(* CODESYS project sortingmachineOOP

Project tree, tasks and I/O mapping:
  Device : CODESYS Control Win V3 x64, 3S - Smart Software Solutions GmbH, version 3.5.16.40
    application Application
      libraries: Standard, * (System); Util, * (System); OMAC PackML State Machine, 1.0.0.4 (3S - Smart Software Solutions GmbH); Alarm Manager Interfaces, * (Intern); SysTypes Interfaces, 3.5.2.0 (System); VisuDialogs, * (System); XML parsing and composing library, * (Open Source); StringUtils, 3.5.17.0 (System); SysMem, 3.5.17.0 (System); CAA File, 3.5.17.0 (CAA Technical Workgroup); CAA Types Extern, 3.5.17.0 (CAA Technical Workgroup); CmpErrors Interfaces, * (System); SysDir, 3.5.17.0 (System); SysFile, 3.5.17.0 (System); SysTimeRtc, 3.5.17.0 (System)
      task AlarmManagerTask (cyclic, interval 50 ms, priority 31) calls AlarmManager.Alarm_Prg
      task MainTask (cyclic, interval t#20ms, priority 1) calls PLC_PRG, Sortery, LogowanieDanych
      task Task (cyclic, interval 5 ms, priority 1) calls POU_cyclic
      task VISU_TASK (cyclic, interval 100 ms, priority 31) calls VisuElems.Visu_Prg
      Alarm Configuration
        alarm group AlarmGroup1
            0 [Error]: Comparison Equal, ExpressionToCompare FALSE, Expression FIO.xEmergencyStop - "Przycisk bezpieczeństwa"
            2 [Warning]: Comparison Equal, ExpressionToCompare TRUE, Expression FIO.xSyrena - "Koniec przerwy"
            3 [Info]: Comparison Equal, ExpressionToCompare PACK_ML.State.Held, Expression PLC_PRG.unitModeManager.ActiveUnitMode.CurrentState - "Maszyna w stanie HELD"
            4 [Info]: Comparison Equal, ExpressionToCompare PACK_ML.State.Suspended, Expression PLC_PRG.unitModeManager.ActiveUnitMode.CurrentState - "Maszyna w stanie SUSPENDED"
            5 [Error]: Comparison Equal, ExpressionToCompare PACK_ML.State.Aborted, Expression PLC_PRG.unitModeManager.ActiveUnitMode.CurrentState - "Maszyna w stanie ABORTED"
        text list AlarmGroup1
        alarm group AlarmGroup2
        text list AlarmGroup2
        alarm group AlarmGroup3
        text list AlarmGroup3
        text list AlarmGroup
        AlarmStorage
        alarm class Error (priority 10, acknowledge ACK_REP_ACK)
        alarm class Info (priority 100, acknowledge REP)
        alarm class Warning (priority 30, acknowledge REP_ACK)
      Alarmy/
        function block AlarmFilterCriteria [ST]: AreAllAlarmClassesSelected, AreAllAlarmGroupsSelected, GetAlarmClasses, GetAlarmGroups, GetCountAlarmClasses, GetCountAlarmGroups, GetPriorityFrom, GetPriorityTo
        function block AlarmManagerClient [ST]: ActiveAlarmsChanged, AfterInit, AlarmStorageModified, GetFilterCriteria
        function ProcessAlarms [ST]
        data type StructureAlarmAsStrings
      Class Diagram
      Czas/
        function PobranieCzasu [ST]
        function UpdateEventTimestampWithSystemTime [ST]
      Data logger/
        data type E_EventSeverity
        data type E_EventType
        data type E_MaxString
        function block FB_CsvPersistentEventStorage [ST]: CreateCsvString, StoreEvent
        function block FB_EventLogger [ST]: AddEvent, FB_Init, IsEventBufferFull
        function block FB_XmlPac [ST]: ComposeXmlExample, FB_Init, OpenWriteClose, Parse, StoreEvent
        data type ST_Event
      data type eKolumnaKolor
      Interfejsy/
        interface I_Kolumna: M_BuzzerOnOff, M_UstawKolor
        interface I_PersistentEventStorage: StoreEvent
        interface I_Przenosnik: MaxPredkosc, MinPredkosc, PredkoscZadana, Start, Stop
      Obiekty/
        function block FB_Kolumna [ST]: M_BuzzerOnOff, M_UstawKolor
        function block FB_Przenosnik [ST]: MaxPredkosc, MinPredkosc, Predkosc, PredkoscZadana, Start, Stop
        function block FB_PrzenosnikNowy [ST]: AktualnaLiczbaZleconychProduktow, ZlecenieProdukty, ZliczajProdukty
        function block Sorter [ST]
        function block Sorter_1 [ST]: Bazowanie, Bazowanie_koniec, Czekaj, Error, FB_Init, Init, Sortowanie, SortowanieKoniec, TRANS_BAZOWANIE, TRANS_BAZOWANIE_KONIEC, TRANS_CZEKAJ, TRANS_ERROR, TRANS_INIT, TRANS_SORTOWANIE, TRANS_SORTOWANIE_KONIEC
      visualisation Panel
      Programy/
        program LogowanieDanych [ST]
        program PLC_PRG [ST]
        program POU_cyclic [ST]
        program Sortery [ST]
      Zmienne globalne/
        global variables FIO
        global variables GVL
    Ethernet : Ethernet, 3S - Smart Software Solutions GmbH, version 3.5.17.0
      Modbus_TCP_Master : Modbus TCP Master, 3S - Smart Software Solutions GmbH, version 3.5.16.0
          settings: AutoReconnect = TRUE
        Modbus_TCP_Slave : Modbus TCP Slave, 3S - Smart Software Solutions GmbH, version 3.5.16.0
            settings: Unit-ID = 1; IPAddress = [127, 0, 0, 1]; Salon_A_FC_02.Function Code = 2; Salon_A_FC_02.Read Offset = 16#0000; Salon_A_FC_02.Read Length = 16; Salon_A_FC_02.Write Offset = 0; Salon_A_FC_02.Write Length = 0; Salon_A_FC_02.Cycle Time = 100; Salon_A_FC_03.Function Code = 4; Salon_A_FC_03.Read Offset = 16#0000; Salon_A_FC_03.Read Length = 8; Salon_A_FC_03.Write Offset = 0; Salon_A_FC_03.Write Length = 0; Salon_A_FC_03.Cycle Time = 20; Salon_A_FC_15.Function Code = 15; Salon_A_FC_15.Read Offset = 0; Salon_A_FC_15.Read Length = 0; Salon_A_FC_15.Write Offset = 16#0000; Salon_A_FC_15.Write Length = 16; Salon_A_FC_15.Cycle Time = 100; Channel 3.Function Code = 16; Channel 3.Read Offset = 0; Channel 3.Read Length = 0; Channel 3.Write Offset = 16#0000; Channel 3.Write Length = 5; Channel 3.Cycle Time = 100
            input  Application.FIO.xPrzyciskStart : BOOL  // Salon_A_FC_02.Salon_A_FC_02.Bit0
            input  Application.FIO.xPrzyciskStop : BOOL  // Salon_A_FC_02.Salon_A_FC_02.Bit1
            input  Application.FIO.xPrzyciskReset : BOOL  // Salon_A_FC_02.Salon_A_FC_02.Bit2
            input  Application.FIO.xEmergencyStop : BOOL  // Salon_A_FC_02.Salon_A_FC_02.Bit3
            input  Application.FIO.xTrybAutoManual : BOOL  // Salon_A_FC_02.Salon_A_FC_02.Bit4
            input  Application.FIO.xCzujnikWejscie : BOOL  // Salon_A_FC_02.Salon_A_FC_02.Bit5
            input  Application.FIO.xCzujnikElementNOK_1 : BOOL  // Salon_A_FC_02.Salon_A_FC_02.Bit6
            input  Application.FIO.xCzujnikElementOK_2 : BOOL  // Salon_A_FC_02.Salon_A_FC_02.Bit7
            input  Application.FIO.xCzujnikElementOK_3 : BOOL  // Salon_A_FC_02.Salon_A_FC_02.Bit0
            input  Application.FIO.xFIOAktywny : BOOL  // Salon_A_FC_02.Salon_A_FC_02.Bit1
            input  Application.FIO.iCzujnikWizyjny : WORD  // Salon_A_FC_03.Salon_A_FC_03
            output Application.FIO.xLampkaStart : BOOL  // Salon_A_FC_15.Salon_A_FC_15.Bit0
            output Application.FIO.xLampkaStop : BOOL  // Salon_A_FC_15.Salon_A_FC_15.Bit1
            output Application.FIO.xLampkaReset : BOOL  // Salon_A_FC_15.Salon_A_FC_15.Bit2
            output Application.FIO.xSorterObroc_1 : BOOL  // Salon_A_FC_15.Salon_A_FC_15.Bit3
            output Application.FIO.xSorterPas_1 : BOOL  // Salon_A_FC_15.Salon_A_FC_15.Bit4
            output Application.FIO.xSorterObroc_2 : BOOL  // Salon_A_FC_15.Salon_A_FC_15.Bit5
            output Application.FIO.xSorterPas_2 : BOOL  // Salon_A_FC_15.Salon_A_FC_15.Bit6
            output Application.FIO.xSorterObroc_3 : BOOL  // Salon_A_FC_15.Salon_A_FC_15.Bit7
            output Application.FIO.xSorterPas_3 : BOOL  // Salon_A_FC_15.Salon_A_FC_15.Bit0
            output Application.FIO.xPrzeslona : BOOL  // Salon_A_FC_15.Salon_A_FC_15.Bit1
            output Application.FIO.xKolumnaLampaCzerwona : BOOL  // Salon_A_FC_15.Salon_A_FC_15.Bit2
            output Application.FIO.xKolumnaLampaZielona : BOOL  // Salon_A_FC_15.Salon_A_FC_15.Bit3
            output Application.FIO.xKolumnaLampaZolta : BOOL  // Salon_A_FC_15.Salon_A_FC_15.Bit4
            output Application.FIO.xKolumnaLampaNiebieski : BOOL  // Salon_A_FC_15.Salon_A_FC_15.Bit5
            output Application.FIO.xEmiter : BOOL  // Salon_A_FC_15.Salon_A_FC_15.Bit6
            output Application.FIO.xSyrena : BOOL  // Salon_A_FC_15.Salon_A_FC_15.Bit7
            output Application.FIO.iPodajnikWejsciowy : WORD  // Channel 3.Channel 3
            output Application.FIO.iPodajnikWyjsciowy : WORD  // Channel 3.Channel 3
            output Application.FIO.iLicznik_1 : WORD  // Channel 3.Channel 3
            output Application.FIO.iLicznik_2 : WORD  // Channel 3.Channel 3
            output Application.FIO.iLicznik_3 : WORD  // Channel 3.Channel 3
            unmapped channels: Salon_A_FC_02, Salon_A_FC_03, Salon_A_FC_15, Channel 3
  text list GlobalTextList
*)

// Device/Application/eKolumnaKolor
{attribute 'qualified_only'}
{attribute 'strict'}
TYPE eKolumnaKolor :
(
	zielony := 0,
	czerwony := 1,
	zolty := 2,
	niebieski := 3
);
END_TYPE

// Device/Application/Alarmy/StructureAlarmAsStrings
/// This structure contains the data the alarm table simulation displays in one row
TYPE StructureAlarmAsStrings :
STRUCT
	sState		: STRING;
	sID			: STRING;
	sInternalID	: STRING;
	sMessage	: STRING;
	sAlarmGroup	: STRING;
	sTSLast		: STRING;
	sAlarmClass	: STRING;
	sPriority	: STRING;
	sCurrValue	: STRING;
	sLatchVar1	: STRING;
	sLatchVar2	: STRING;
END_STRUCT
END_TYPE

// Device/Application/Data logger/E_EventSeverity
{attribute 'qualified_only'}
{attribute 'strict'}
TYPE E_EventSeverity :
(
    Verbose  := 0, // in progress
    Info     := 1, 
    Warning  := 2, 
    Error    := 3, 
    Critical := 4);
END_TYPE

// Device/Application/Data logger/E_EventType
{attribute 'qualified_only'}
{attribute 'strict'}
{attribute 'to_string'}
TYPE E_EventType :
(
	Alarm := 0,
	Message := 1
);
END_TYPE

// Device/Application/Data logger/E_MaxString
{attribute 'qualified_only'}
{attribute 'strict'}
TYPE E_MaxString :
(
	MaxString := 255
);
END_TYPE

// Device/Application/Data logger/ST_Event
TYPE ST_Event :
STRUCT
	eEventType : E_EventType;
	eEventSeverity: E_EventSeverity;
	nEventIdentity : UDINT;
	sEventText : STRING(255);
	dtTimeStamp: DATE_AND_TIME;
END_STRUCT

END_TYPE

// Device/Application/Zmienne globalne/FIO
{attribute 'qualified_only'}
VAR_GLOBAL
	(* zmienne wejściowe *)
	xPrzyciskStart:BOOL; // Start przenośnika - wejście PLC
	xPrzyciskStop:BOOL; // Stop przenośnika - wejście PLC
	xPrzyciskReset: BOOL; // Reset maszyny
	xEmergencyStop: BOOL; // Stop awaryjny
	xTrybAutoManual: BOOL; // Przełącznik piórkowy, mtryb auto/manual
	xCzujnikWejscie: BOOL; // czujnik na linii wejściowej
	xCzujnikElementNOK_1: BOOL; // wykrywa elementy wadliwe na linii, zsuwnia pierwsza
	xCzujnikElementOK_2: BOOL; // wykrywa elementy poprawne, zsuwnia druga
	xCzujnikElementOK_3: BOOL; //  wykrywa elementy poprawne, zsuwnia trzecia
	xFIOAktywny: BOOL;
	
	
	iCzujnikWizyjny: INT; // zwraca wartości ID poszczególnych elementów na linii
	
	(* zmienne wyjściowe *)
	xLampkaStart:BOOL; // podświetlenie przycisku start
	xLampkaStop:BOOL; // podśwoetlenie przycisku stop
	xLampkaReset: BOOL; // podśwoetlenie przycisku reet
	xSorterObroc_1: BOOL; // sorter spychający wadliwe elementy do zsuwni, sorter 1
	xSorterPas_1: BOOL; // pas sortera nr 1
	xSorterObroc_2: BOOL; // sorter spychający prawidłowe elementy do zsuwni, sorter 2
	xSorterPas_2: BOOL; // pas sortera nr 2
	xSorterObroc_3: BOOL; // sorter spychający prawidłowe elementy do zsuwni, sorter 3
	xSorterPas_3: BOOL; // pas sortera nr 3
	xPrzeslona: BOOL; // przesłona między podajnikami
	xSyrena:BOOL; // Syrena na przenośniku
	xKolumnaLampaCzerwona: BOOL; //  czerwona lampa kolumna świetlna
	xKolumnaLampaZielona: BOOL; //  zielona lampa kolumna świetlna
	xKolumnaLampaZolta: BOOL; //  zółta lampa kolumna świetlna
	xKolumnaLampaNiebieski : BOOL; //  niebeiska lampka kolumna świetlna
	xSorterLampa_1 :BOOL; // sygnalizacja świetlna sortera nr 1
	xSorterLampa_2 :BOOL; // sygnalizacja świetlna sortera nr 2
	xSorterLampa_3 :BOOL; // sygnalizacja świetlna sortera nr 3
	xEmiter: bool; // generator elementów na liniii
	
	iPodajnikWejsciowy: INT; // wpisujemy wartośc od 0-1000 w celu regulacji prędkości podajnika
	iPodajnikWyjsciowy: INT; // wpisujemy wartośc od 0-1000 w celu regulacji prędkości podajnika
	iLicznik_1: INT; 
	iLicznik_2: INT;
	iLicznik_3: INT;

END_VAR

// Device/Application/Zmienne globalne/GVL
{attribute 'qualified_only'}
VAR_GLOBAL
	xErrorActive:BOOL:=0;
	aAlarmy: ARRAY [0..19] OF BOOL; 	// tablica alarmów, klasa Error
	wAlarmy: WORD:=0;
	xResetAlarm: BOOL;
	g_sAlarmID:STRING;
    aRejestrProduktow : ARRAY[0..100] OF DINT;
    diSensorWizyjnyOstatniaWartosc : DINT;
    xLiniaStart : BOOL;
    xAlarmAktywny : BOOL;
	R_TRIG_Start:R_TRIG;
	R_TRIG_Reset:F_TRIG; 
	g_sMainDirectory : STRING := 'c:/'; // ścieżka głowna pliku CSV dla data logger
END_VAR
VAR_GLOBAL CONSTANT
	{attribute 'const_replaced'}
	gc_iNoOfCollumns:INT :=15;
	gc_iLengthOfDataArray:INT:=255;
	
	// PackML
	gc_sPRODUCTION : STRING := 'Production';
	gc_sSEMIAUTO : STRING := 'Semi Auto';
	gc_sSETUP : STRING := 'Setup';
END_VAR

// Device/Application/Programy/PLC_PRG
PROGRAM PLC_PRG
VAR
	productionUnitMode	: PACK_ML.UnitMode; // Example unit mode for prodction
	semiAutoUnitMode	: PACK_ML.UnitMode; // Example unit mode for semi auto production
	setupUnitMode		: PACK_ML.UnitMode; // Example unit mode for setup
	unitModeManager		: PACK_ML.UnitModeManager; // Unit mode manager to switch between unitmodes
	currentUnitMode		: PACK_ML.IUnitMode;
	xInit				: BOOL := FALSE; // Flag for initialization	
	
	// Visu Commands	
	xAbort				: BOOL;
	xActingStateComplete: BOOL;
	xClear				: BOOL;
	xHold				: BOOL;
	xReset				: BOOL;
	xStart				: BOOL;
	xStop				: BOOL;
	xSuspend			: BOOL;
	xUnHold				: BOOL;
	xUnSuspend			: BOOL;
	
	// Helper
	xSimulate			: BOOL;
	xChangeState		: BOOL := FALSE;	
	timer1				: TON;	
	iSelectedUnitMode	: INT := 0;
	iLastSelectedUnitMode: INT := 0;
	xUserModeChanged	: BOOL;
	xTest: BOOL;
	itest: INT;
	
	fbPrzenosnik: FB_PrzenosnikNowy;
	
	// alarm manager
	mAlarmManagerClient: AlarmManagerClient;
	
	StartStop: RS;
	xZlecenieWykonane: BOOL;
	LicznikElementyNaLinii: CTUD;
	iMaxPredkosc_visu: INT;
	iMinPredkosc_visu: INT;
	iPredkoscZadana_visu: INT;
	iZlecenie_visu: INT;
	xPotwierdzParametry_visu: BOOL;
	
	fbRtrigCzujnikSorter_1: r_trig;
	fbRtrigCzujnikSorter_2: r_trig;
	fbRtrigCzujnikSorter_3: r_trig;
	xResetZlecenie_visu: BOOL;
	iAktualnaLiczbaZleconychProduktow_visu: INT;
	fbKolumna: FB_Kolumna;
END_VAR

// inicjalizacja trybu pracy w standardzie Pack ML
IF NOT xInit THEN
	productionUnitMode(		sName := gvl.gc_sPRODUCTION, 
							dwSupportedStates := PACK_ML.State.All, 
							dwAllowsLeavingFromStates := PACK_ML.State.Stopped OR PACK_ML.State.Aborted OR PACK_ML.State.Idle, 
							dwAllowsEnteringIntoStates := PACK_ML.State.Stopped OR PACK_ML.State.Aborted OR PACK_ML.State.Idle, 
							eInitialState := PACK_ML.State.Resetting,
							xActive := TRUE);
	semiAutoUnitMode(		sName := gvl.gc_sSEMIAUTO, 
							dwSupportedStates := PACK_ML.State.All - PACK_ML.State.Completing - PACK_ML.State.Complete - PACK_ML.State.Holding - PACK_ML.State.Held - PACK_ML.State.UnHolding,
							dwAllowsLeavingFromStates := PACK_ML.State.Stopped OR PACK_ML.State.Aborted OR PACK_ML.State.Idle, 
							dwAllowsEnteringIntoStates := PACK_ML.State.Stopped OR PACK_ML.State.Aborted OR PACK_ML.State.Idle,   
							eInitialState := PACK_ML.State.Idle, 
							xActive := FALSE);
	setupUnitMode(			sName := gvl.gc_sSETUP, 
							dwSupportedStates := PACK_ML.State.All - PACK_ML.State.Completing - PACK_ML.State.Complete - PACK_ML.State.Holding - PACK_ML.State.Held - PACK_ML.State.UnHolding - PACK_ML.State.UnSuspending - PACK_ML.State.Suspended - PACK_ML.State.Suspending,
							dwAllowsLeavingFromStates := PACK_ML.State.Stopped OR PACK_ML.State.Aborted OR PACK_ML.State.Idle,   
							dwAllowsEnteringIntoStates := PACK_ML.State.Stopped OR PACK_ML.State.Aborted OR PACK_ML.State.Idle, 
							eInitialState := PACK_ML.State.Idle, 
							xActive := FALSE);
	
	// inicjalizacja wartości dla maszyny
	fbPrzenosnik.MaxPredkosc := 10;
	fbPrzenosnik.MinPredkosc := 2;
	fbPrzenosnik.PredkoscZadana := 4;
			

	// Register the unit modes 
	unitModeManager.Register(productionUnitMode);
	unitModeManager.Register(semiAutoUnitMode);
	unitModeManager.Register(setupUnitMode);
	xInit := TRUE;
END_IF

IF FIO.xFIOAktywny THEN
	
mAlarmManagerClient();

fbKolumna();

// wywołanie instancji przenośnika
fbPrzenosnik(in_xEnable:= TRUE, out_iSilnik=> fio.iPodajnikWejsciowy);
fio.iPodajnikWyjsciowy := fio.iPodajnikWejsciowy;

fbRtrigCzujnikSorter_1(CLK:= NOT FIO.xCzujnikElementOK_3, Q=> );
fbRtrigCzujnikSorter_2(CLK:= NOT FIO.xCzujnikElementOK_2 , Q=> );
fbRtrigCzujnikSorter_3(CLK:= NOT FIO.xCzujnikElementNOK_1 , Q=> );



// Zmiana trybu pracy jednostki Pack ML
IF iSelectedUnitMode <> iLastSelectedUnitMode THEN
	IF iSelectedUnitMode = 0 THEN
		xUserModeChanged := unitModeManager.SwitchUnitMode(gvl.gc_sPRODUCTION);
	ELSIF iSelectedUnitMode = 1 THEN
		xUserModeChanged := unitModeManager.SwitchUnitMode(gvl.gc_sSEMIAUTO);
	ELSE
 		xUserModeChanged := unitModeManager.SwitchUnitMode(gvl.gc_sSETUP);
	END_IF
	IF xUserModeChanged THEN
		iLastSelectedUnitMode := iSelectedUnitMode;
	ELSE
		iSelectedUnitMode := iLastSelectedUnitMode;
	END_IF
END_IF

// Sprawdzenie czy jednostka aktywna
IF unitModeManager.ActiveUnitMode <> 0 THEN	
	currentUnitMode := unitModeManager.ActiveUnitMode;
	
	IF  NOT fio.xEmergencyStop THEN
		unitModeManager.ActiveUnitMode.Abort();
	END_IF
	
	IF NOT fio.xPrzyciskStop OR xStop THEN
		GVL.xLiniaStart := FALSE;
		unitModeManager.ActiveUnitMode.Stop();
	END_IF
	
	// sekwencja Pack ML
	CASE unitModeManager.ActiveUnitMode.CurrentState OF
		PACK_ML.State.Stopped:
			fbKolumna.M_BuzzerOnOff(in_xOnOff:= FALSE, out_xBuzzer=> fio.xSyrena );
			fbKolumna.M_UstawKolor(in_xEnable:= TRUE, in_iKolor:= eKolumnaKolor.czerwony, in_xImpusatorOnOff:= FALSE, 
								  out_xZielony=> fio.xKolumnaLampaZielona, out_xCzerwony=> fio.xKolumnaLampaCzerwona, out_xZolty=> fio.xKolumnaLampaZolta, out_xNiebieski=> fio.xKolumnaLampaNiebieski );
			IF fio.xPrzyciskReset OR xReset THEN
				unitModeManager.ActiveUnitMode.Reset(); // przejście do kolejnego stanu
			END_IF;
			
		PACK_ML.State.Resetting:	
			fbKolumna.M_BuzzerOnOff(in_xOnOff:= FALSE, out_xBuzzer=> fio.xSyrena );
			fbKolumna.M_UstawKolor(in_xEnable:= TRUE, in_iKolor:= eKolumnaKolor.czerwony, in_xImpusatorOnOff:= FALSE, 
								  out_xZielony=> fio.xKolumnaLampaZielona, out_xCzerwony=> fio.xKolumnaLampaCzerwona, out_xZolty=> fio.xKolumnaLampaZolta, out_xNiebieski=> fio.xKolumnaLampaNiebieski );
			fbPrzenosnik.MaxPredkosc := iMaxPredkosc_visu;
			fbPrzenosnik.MinPredkosc := iMinPredkosc_visu;
			fbPrzenosnik.PredkoscZadana := iPredkoscZadana_visu;
			
			fbPrzenosnik.ZliczajProdukty(in_xResetZlecenia:= xResetZlecenie_visu, in_xLicznikElementow:= fbRtrigCzujnikSorter_1.Q OR fbRtrigCzujnikSorter_2.Q OR fbRtrigCzujnikSorter_3.Q);
			iAktualnaLiczbaZleconychProduktow_visu := fbPrzenosnik.AktualnaLiczbaZleconychProduktow;
			
			IF fbPrzenosnik.AktualnaLiczbaZleconychProduktow = 0 THEN
				fbPrzenosnik.ZlecenieProdukty := iZlecenie_visu;
			END_IF
			
			IF ( fbPrzenosnik.MinPredkosc <> 0 AND  
				fbPrzenosnik.MaxPredkosc <> 0 AND 
				fbPrzenosnik.ZlecenieProdukty <> 0 AND 
				fbPrzenosnik.PredkoscZadana <> 0 AND 
				xPotwierdzParametry_visu ) 
			THEN
				unitModeManager.ActiveUnitMode.ActingStateCompleted(); // przejście do stanu IDLE
			END_IF;
					
		PACK_ML.State.Idle:	
			fbKolumna.M_BuzzerOnOff(in_xOnOff:= FALSE, out_xBuzzer=> fio.xSyrena );
			fbKolumna.M_UstawKolor(in_xEnable:= TRUE, in_iKolor:= eKolumnaKolor.zielony, in_xImpusatorOnOff:= TRUE, 
								  out_xZielony=> fio.xKolumnaLampaZielona, out_xCzerwony=> fio.xKolumnaLampaCzerwona, out_xZolty=> fio.xKolumnaLampaZolta, out_xNiebieski=> fio.xKolumnaLampaNiebieski );		

			fio.xEmiter := TRUE;
			IF fio.xPrzyciskStart OR xStart THEN
				unitModeManager.ActiveUnitMode.Start();
			END_IF
			
		PACK_ML.State.Starting:
			fbKolumna.M_BuzzerOnOff(in_xOnOff:= FALSE, out_xBuzzer=> fio.xSyrena );
			fbKolumna.M_UstawKolor(in_xEnable:= TRUE, in_iKolor:= eKolumnaKolor.zielony, in_xImpusatorOnOff:= FALSE, 
								  out_xZielony=> fio.xKolumnaLampaZielona, out_xCzerwony=> fio.xKolumnaLampaCzerwona, out_xZolty=> fio.xKolumnaLampaZolta, out_xNiebieski=> fio.xKolumnaLampaNiebieski );		


			fbPrzenosnik.Start(1); //  metoda start z parametrem iRampa ( przedział 1-10)
			GVL.xLiniaStart := TRUE;
			IF fbPrzenosnik.out_iSilnik = fbPrzenosnik.PredkoscZadana THEN
				unitModeManager.ActiveUnitMode.ActingStateCompleted(); // przejście do stanu EXECUTE
			END_IF
			
		PACK_ML.State.Execute:	
			fbKolumna.M_BuzzerOnOff(in_xOnOff:= FALSE, out_xBuzzer=> fio.xSyrena );
			fbKolumna.M_UstawKolor(in_xEnable:= TRUE, in_iKolor:= eKolumnaKolor.zielony, in_xImpusatorOnOff:= FALSE, 
								  out_xZielony=> fio.xKolumnaLampaZielona, out_xCzerwony=> fio.xKolumnaLampaCzerwona, out_xZolty=> fio.xKolumnaLampaZolta, out_xNiebieski=> fio.xKolumnaLampaNiebieski );			
			fbPrzenosnik.ZliczajProdukty(in_xLicznikElementow:= fbRtrigCzujnikSorter_1.Q OR fbRtrigCzujnikSorter_2.Q OR fbRtrigCzujnikSorter_3.Q, in_xResetZlecenia:= xResetZlecenie_visu);
			
			IF xHold THEN
				unitModeManager.ActiveUnitMode.Hold();
			END_IF
			
			IF xSuspend THEN
				unitModeManager.ActiveUnitMode.Suspend();
			END_IF
			
			iAktualnaLiczbaZleconychProduktow_visu := fbPrzenosnik.AktualnaLiczbaZleconychProduktow;
			
			IF fbPrzenosnik.AktualnaLiczbaZleconychProduktow = fbPrzenosnik.ZlecenieProdukty THEN
				unitModeManager.ActiveUnitMode.ActingStateCompleted();
			END_IF
						
		PACK_ML.State.Holding:
			fbKolumna.M_BuzzerOnOff(in_xOnOff:= FALSE, out_xBuzzer=> fio.xSyrena );
			fbKolumna.M_UstawKolor(in_xEnable:= TRUE, in_iKolor:= eKolumnaKolor.niebieski, in_xImpusatorOnOff:= FALSE, 
								  out_xZielony=> fio.xKolumnaLampaZielona, out_xCzerwony=> fio.xKolumnaLampaCzerwona, out_xZolty=> fio.xKolumnaLampaZolta, out_xNiebieski=> fio.xKolumnaLampaNiebieski );		
				fbPrzenosnik.Stop();
				unitModeManager.ActiveUnitMode.ActingStateCompleted();
				
		PACK_ML.State.Held:
			fbKolumna.M_BuzzerOnOff(in_xOnOff:= FALSE, out_xBuzzer=> fio.xSyrena );
			fbKolumna.M_UstawKolor(in_xEnable:= TRUE, in_iKolor:= eKolumnaKolor.niebieski, in_xImpusatorOnOff:= FALSE, 
								  out_xZielony=> fio.xKolumnaLampaZielona, out_xCzerwony=> fio.xKolumnaLampaCzerwona, out_xZolty=> fio.xKolumnaLampaZolta, out_xNiebieski=> fio.xKolumnaLampaNiebieski );		
			IF xUnHold THEN
				unitModeManager.ActiveUnitMode.UnHold();
			END_IF
				
		PACK_ML.State.UnHolding:
			fbKolumna.M_BuzzerOnOff(in_xOnOff:= FALSE, out_xBuzzer=> fio.xSyrena );
			fbKolumna.M_UstawKolor(in_xEnable:= TRUE, in_iKolor:= eKolumnaKolor.niebieski, in_xImpusatorOnOff:= TRUE, 
								  out_xZielony=> fio.xKolumnaLampaZielona, out_xCzerwony=> fio.xKolumnaLampaCzerwona, out_xZolty=> fio.xKolumnaLampaZolta, out_xNiebieski=> fio.xKolumnaLampaNiebieski );		


			fbPrzenosnik.Start(fbPrzenosnik.PredkoscZadana); 
			IF fbPrzenosnik.Predkosc > 0 THEN
				unitModeManager.ActiveUnitMode.ActingStateCompleted();
			END_IF
	
			
		PACK_ML.State.Suspending:
			fbKolumna.M_BuzzerOnOff(in_xOnOff:= FALSE, out_xBuzzer=> fio.xSyrena );
			fbKolumna.M_UstawKolor(in_xEnable:= TRUE, in_iKolor:= eKolumnaKolor.zolty, in_xImpusatorOnOff:= TRUE, 
								  out_xZielony=> fio.xKolumnaLampaZielona, out_xCzerwony=> fio.xKolumnaLampaCzerwona, out_xZolty=> fio.xKolumnaLampaZolta, out_xNiebieski=> fio.xKolumnaLampaNiebieski );		
			fbPrzenosnik.Stop();
			unitModeManager.ActiveUnitMode.ActingStateCompleted();
				
		PACK_ML.State.Suspended:
			fbKolumna.M_BuzzerOnOff(in_xOnOff:= TRUE, out_xBuzzer=> fio.xSyrena );
			fbKolumna.M_UstawKolor(in_xEnable:= TRUE, in_iKolor:= eKolumnaKolor.zolty, in_xImpusatorOnOff:= TRUE, 
								  out_xZielony=> fio.xKolumnaLampaZielona, out_xCzerwony=> fio.xKolumnaLampaCzerwona, out_xZolty=> fio.xKolumnaLampaZolta, out_xNiebieski=> fio.xKolumnaLampaNiebieski );		


			IF xUnSuspend THEN
				unitModeManager.ActiveUnitMode.UnSuspend();
			END_IF
			
		PACK_ML.State.UnSuspending:
			fbKolumna.M_BuzzerOnOff(in_xOnOff:= FALSE, out_xBuzzer=> fio.xSyrena );
			fbKolumna.M_UstawKolor(in_xEnable:= TRUE, in_iKolor:= eKolumnaKolor.niebieski, in_xImpusatorOnOff:= TRUE, 
								  out_xZielony=> fio.xKolumnaLampaZielona, out_xCzerwony=> fio.xKolumnaLampaCzerwona, out_xZolty=> fio.xKolumnaLampaZolta, out_xNiebieski=> fio.xKolumnaLampaNiebieski );		

				fbPrzenosnik.Start(fbPrzenosnik.PredkoscZadana);
				IF fbPrzenosnik.Predkosc > 0 THEN
					unitModeManager.ActiveUnitMode.ActingStateCompleted();
				END_IF
				
		PACK_ML.State.Completing:
			fbKolumna.M_BuzzerOnOff(in_xOnOff:= FALSE, out_xBuzzer=> fio.xSyrena );
			fbKolumna.M_UstawKolor(in_xEnable:= TRUE, in_iKolor:= eKolumnaKolor.zielony, in_xImpusatorOnOff:= FALSE, 
								  out_xZielony=> fio.xKolumnaLampaZielona, out_xCzerwony=> fio.xKolumnaLampaCzerwona, out_xZolty=> fio.xKolumnaLampaZolta, out_xNiebieski=> fio.xKolumnaLampaNiebieski );		

			fbPrzenosnik.Stop();
			unitModeManager.ActiveUnitMode.ActingStateCompleted();
			
		PACK_ML.State.Complete:	
			fbKolumna.M_BuzzerOnOff(in_xOnOff:= FALSE, out_xBuzzer=> fio.xSyrena );
			fbKolumna.M_UstawKolor(in_xEnable:= TRUE, in_iKolor:= eKolumnaKolor.czerwony, in_xImpusatorOnOff:= FALSE, 
								  out_xZielony=> fio.xKolumnaLampaZielona, out_xCzerwony=> fio.xKolumnaLampaCzerwona, out_xZolty=> fio.xKolumnaLampaZolta, out_xNiebieski=> fio.xKolumnaLampaNiebieski );		
	
			IF xReset THEN
				unitModeManager.ActiveUnitMode.Reset();
			END_IF
			
		PACK_ML.State.Stopping:
			fbKolumna.M_BuzzerOnOff(in_xOnOff:= FALSE, out_xBuzzer=> fio.xSyrena );
			fbKolumna.M_UstawKolor(in_xEnable:= TRUE, in_iKolor:= eKolumnaKolor.czerwony, in_xImpusatorOnOff:= FALSE, 
								  out_xZielony=> fio.xKolumnaLampaZielona, out_xCzerwony=> fio.xKolumnaLampaCzerwona, out_xZolty=> fio.xKolumnaLampaZolta, out_xNiebieski=> fio.xKolumnaLampaNiebieski );		

			fio.xEmiter := FALSE;
		
		PACK_ML.State.Aborting:
			fbKolumna.M_BuzzerOnOff(in_xOnOff:= FALSE, out_xBuzzer=> fio.xSyrena );
			fbKolumna.M_UstawKolor(in_xEnable:= TRUE, in_iKolor:= eKolumnaKolor.czerwony, in_xImpusatorOnOff:= TRUE, 
								  out_xZielony=> fio.xKolumnaLampaZielona, out_xCzerwony=> fio.xKolumnaLampaCzerwona, out_xZolty=> fio.xKolumnaLampaZolta, out_xNiebieski=> fio.xKolumnaLampaNiebieski );		

				fbPrzenosnik.Stop();
				GVL.xLiniaStart := FALSE;
				unitModeManager.ActiveUnitMode.ActingStateCompleted();
		PACK_ML.State.Aborted:
			fbKolumna.M_BuzzerOnOff(in_xOnOff:= FALSE, out_xBuzzer=> fio.xSyrena );
			fbKolumna.M_UstawKolor(in_xEnable:= TRUE, in_iKolor:= eKolumnaKolor.czerwony, in_xImpusatorOnOff:= TRUE, 
								  out_xZielony=> fio.xKolumnaLampaZielona, out_xCzerwony=> fio.xKolumnaLampaCzerwona, out_xZolty=> fio.xKolumnaLampaZolta, out_xNiebieski=> fio.xKolumnaLampaNiebieski );		
		
			IF  NOT (mAlarmManagerClient.out_aAlarmsAsStrings[0].sState = 'Active')  (* OR  mAlarmManagerClient.out_aAlarmsAsStrings[0].sState = 'ActiveAcknowledged' *)  THEN
				IF xClear THEN
					unitModeManager.ActiveUnitMode.Clear(); // przejście do stanu CLEAR
				END_IF
			END_IF;
		
		PACK_ML.State.Clearing:
			fbKolumna.M_BuzzerOnOff(in_xOnOff:= FALSE, out_xBuzzer=> fio.xSyrena );
			fbKolumna.M_UstawKolor(in_xEnable:= TRUE, in_iKolor:= eKolumnaKolor.czerwony, in_xImpusatorOnOff:= TRUE, 
								  out_xZielony=> fio.xKolumnaLampaZielona, out_xCzerwony=> fio.xKolumnaLampaCzerwona, out_xZolty=> fio.xKolumnaLampaZolta, out_xNiebieski=> fio.xKolumnaLampaNiebieski );		
			IF mAlarmManagerClient.out_aAlarmsAsStrings[0].sState = ''  THEN
				unitModeManager.ActiveUnitMode.ActingStateCompleted();
			END_IF
	END_CASE

END_IF

END_IF

END_PROGRAM

// Device/Application/Obiekty/FB_PrzenosnikNowy
FUNCTION_BLOCK FB_PrzenosnikNowy EXTENDS FB_Przenosnik
VAR_INPUT
END_VAR
VAR_OUTPUT
END_VAR
VAR
	iLicznikElementyLokalnie: INT;
	iZlecenieLokalnie: INT;
END_VAR

SUPER^();

PROPERTY PUBLIC AktualnaLiczbaZleconychProduktow : INT
GET
AktualnaLiczbaZleconychProduktow := iLicznikElementyLokalnie;
END_GET
END_PROPERTY

PROPERTY PUBLIC ZlecenieProdukty : INT
GET
ZlecenieProdukty := iZlecenieLokalnie;
END_GET
SET
iZlecenieLokalnie := ZlecenieProdukty;
END_SET
END_PROPERTY

METHOD PUBLIC ZliczajProdukty : INT
VAR_INPUT
	in_xLicznikElementow: BOOL;
	in_xResetZlecenia: BOOL;
END_VAR
IF in_xLicznikElementow THEN
	iLicznikElementyLokalnie := iLicznikElementyLokalnie + 1;
END_IF

IF in_xResetZlecenia THEN
	iLicznikElementyLokalnie := 0;
END_IF

ZliczajProdukty := iLicznikElementyLokalnie;
END_METHOD

END_FUNCTION_BLOCK

// Device/Application/Obiekty/FB_Przenosnik
FUNCTION_BLOCK FB_Przenosnik IMPLEMENTS I_Przenosnik
VAR_INPUT 
 in_xEnable : BOOL;
END_VAR

VAR_OUTPUT 
  out_iSilnik: INT;
END_VAR

VAR 
	ImpulsatorRampa: blink;
	rtrigrampa: r_trig;
	
	// predkości przenośnika
	iMaxPredkoscLokalna: INT;
	iMinPredkoscLokalna: INT;
	iPredkoscLokalna: INT;
END_VAR

// metoda start
// impuls danych co 10s
ImpulsatorRampa(ENABLE:= TRUE, TIMELOW:= T#100MS, TIMEHIGH:= T#100MS, OUT=> );
rtrigrampa(CLK:= ImpulsatorRampa.OUT);

{warning 'Add property implementation'}
PROPERTY MaxPredkosc : INT
GET
MaxPredkosc := iMaxPredkoscLokalna;
END_GET
SET
iMaxPredkoscLokalna := MaxPredkosc;
END_SET
END_PROPERTY

{warning 'Add property implementation'}
PROPERTY MinPredkosc : INT
GET
MinPredkosc := iMinPredkoscLokalna;
END_GET
SET
iMinPredkoscLokalna := MinPredkosc;
END_SET
END_PROPERTY

PROPERTY Predkosc : INT
GET
Predkosc := out_iSilnik;
END_GET
END_PROPERTY

{warning 'Add property implementation'}
PROPERTY PredkoscZadana : INT
GET
PredkoscZadana := iPredkoscLokalna;
END_GET
SET
iPredkoscLokalna := PredkoscZadana;
END_SET
END_PROPERTY

{warning 'Add method implementation '}
METHOD Start
VAR_INPUT
	in_iRampa: INT ;
END_VAR
IF in_iRampa >= 10 THEN
	in_irampa := 10;
END_IF

IF in_iRampa < 1 THEN
	in_iRampa := 1;
END_IF

IF rtrigrampa.Q THEN
	IF out_iSilnik <= PredkoscZadana THEN
		out_iSilnik := out_iSilnik + in_iRampa;		
	ELSE
		out_iSilnik := PredkoscZadana;
	END_IF
END_IF;
END_METHOD

{warning 'Add method implementation '}
METHOD Stop
out_iSilnik := 0;
END_METHOD

END_FUNCTION_BLOCK

// Device/Application/Interfejsy/I_Przenosnik
INTERFACE I_Przenosnik

PROPERTY MaxPredkosc : INT
GET
END_GET
SET
END_SET
END_PROPERTY

PROPERTY MinPredkosc : INT
GET
END_GET
SET
END_SET
END_PROPERTY

PROPERTY PredkoscZadana : INT
GET
END_GET
SET
END_SET
END_PROPERTY

METHOD Start
VAR_INPUT
	in_iRampa: INT;
END_VAR
END_METHOD

METHOD Stop
VAR_INPUT
END_VAR
END_METHOD

END_INTERFACE

// Device/Application/Alarmy/AlarmManagerClient
{attribute 'call_after_init'}
FUNCTION_BLOCK AlarmManagerClient IMPLEMENTS AlarmManager.IAlarmManagerClient
VAR_INPUT
END_VAR
VAR_OUTPUT
	out_aAlarmsAsStrings: ARRAY[0 .. MAX_ALARMS_COUNT - 1] OF StructureAlarmAsStrings;
END_VAR
VAR CONSTANT
	MAX_ALARMS_COUNT: UINT := 10;
	FILTRED_GROUPS_COUNT: UINT := 2;
END_VAR
VAR
	eStan: (CZEKAJ_NA_POTWIERDZENIE, KASUJ, ACTIVE, ACTIVEACKNOWLEDGED);
	rtrigEstopKasuj: r_trig;
	rs1:rs;
	aAlarmsAsStrings: ARRAY[0 .. MAX_ALARMS_COUNT - 1] OF StructureAlarmAsStrings;
	aStoredAlarmsAsStrings: ARRAY[0 .. MAX_ALARMS_COUNT - 1] OF StructureAlarmAsStrings;

	// Filter and Params
	mAlarmFilterCriteria: AlarmFilterCriteria;
	aFilteredAlarmGroupIDs : ARRAY [0 .. FILTRED_GROUPS_COUNT - 1] OF UDINT := [
		Alm_AlarmConfiguration_Alarmgroup_InternalIDs.ID_AlarmGroup1,
		Alm_AlarmConfiguration_Alarmgroup_InternalIDs.ID_AlarmGroup3
	];
	
	
	aStoredAlarms		: ARRAY [0 .. MAX_ALARMS_COUNT - 1] OF Alarm;
	aitfStoredAlarms	: ARRAY [0 .. MAX_ALARMS_COUNT - 1] OF IAlarm2;
	
	bRowIDValid: BOOL;
	diRowID: DINT;
	xtest: BOOL;
	iTest: INT;
	xTest1: BOOL;
END_VAR

// rtrigEstopKasuj(clk := aAlarmsAsStrings[0].sState = '');
// rs1(SET:= rtrigEstopKasuj.Q, RESET1:= xtest, Q1=> xTest1);

out_aAlarmsAsStrings := aAlarmsAsStrings;


(* Notification by the alarm manager, that the list of active alarms has changed..
 The IAlarmManagerClient instance can retrieve the list of active alarms by
 calling IAlarmHandler2.GetActiveAlarms.*)
METHOD ActiveAlarmsChanged
VAR
	apAlarms: POINTER TO ARRAY[0..0] OF iAlarm;
	iCountAlarms: INT;
	i: INT;
	pStr: POINTER TO STRING;
END_VAR

g_AlarmHandler.GetActiveAlarms( THIS^, parritfActiveAlarms => apAlarms, iCountActiveAlarms => iCountAlarms);

SysMemSet(ADR(aAlarmsAsStrings), 0, SIZEOF(aAlarmsAsStrings));
IF iCountAlarms > 0 THEN
	ProcessAlarms(
		pitfAlarms := apAlarms,
		udiCountAlarms := INT_TO_UDINT(iCountAlarms),
		pAlarmsAsString := ADR(aAlarmsAsStrings),
		udiCountAlarmsAsString := MAX_ALARMS_COUNT
	);
END_IF
END_METHOD

{attribute 'call_after_init'}
METHOD AfterInit : BOOL
VAR_INPUT
END_VAR
VAR
	i: UINT;
END_VAR
mAlarmFilterCriteria.pudiAlarmGroupIDs := ADR(aFilteredAlarmGroupIDs);
mAlarmFilterCriteria.iCountAlarmGroups := UINT_TO_INT(FILTRED_GROUPS_COUNT);

FOR i := 0 TO MAX_ALARMS_COUNT - 1 DO
	aitfStoredAlarms[i] := aStoredAlarms[i];
END_FOR

g_AlarmHandler.RegisterClient(THIS^, ADR(aitfStoredAlarms), UINT_TO_INT(MAX_ALARMS_COUNT));
END_METHOD


(* Notification by the alarm manager, that something in the alarm storage has been
 modified, i.e. a new alarm has been added to the alarm storage or an already
 stored alarm has been modified.*)
METHOD AlarmStorageModified
VAR
	
	iCountRows : INT;
END_VAR

g_AlarmHandler.GetAlarmsFromStorage(
	THIS^,
	iSkipRows := 0,
	bRowIDValid := bRowIDValid,
	diRowID := diRowID,
	iCountRows => iCountRows
);

SysMemSet(ADR(aStoredAlarmsAsStrings), 0, SIZEOF(aStoredAlarmsAsStrings));
IF iCountRows > 0 THEN
	ProcessAlarms(
		pitfAlarms := ADR(aitfStoredAlarms),
		udiCountAlarms := INT_TO_UDINT(iCountRows),
		pAlarmsAsString := ADR(aStoredAlarmsAsStrings),
		udiCountAlarmsAsString := MAX_ALARMS_COUNT
	);
END_IF
END_METHOD

(* Returns an instance of IAlarmFilterCriteria describing the filter criteria
 used to retrieve the currently active alarms or the historic alarms.*)
METHOD GetFilterCriteria : AlarmManager.IAlarmFilterCriteria
GetFilterCriteria := mAlarmFilterCriteria;
END_METHOD

END_FUNCTION_BLOCK

// Device/Application/Alarmy/AlarmFilterCriteria
FUNCTION_BLOCK AlarmFilterCriteria IMPLEMENTS AlarmManager.IAlarmFilterCriteria
VAR_INPUT
	pudiAlarmGroupIDs : POINTER TO ARRAY [0..0] OF UDINT;
	iCountAlarmGroups : INT;
END_VAR
VAR_OUTPUT
END_VAR

(* Indicates, whether there is no explicit selection of alarm classes present, but all alarm classes have been selected*)
METHOD AreAllAlarmClassesSelected : BOOL
AreAllAlarmClassesSelected := TRUE;
END_METHOD

(* Indicates, whether there is no explicit selection of alarm groups present, but all alarm groups have been selected*)
METHOD AreAllAlarmGroupsSelected : BOOL
AreAllAlarmGroupsSelected := pudiAlarmGroupIDs = 0 OR iCountAlarmGroups = 0;
END_METHOD

{warning 'Add method implementation '}
(* Returns the explicitely selected alarm classes. The array contains the internal IDs of the alarm classes to consider.*)
METHOD GetAlarmClasses : POINTER TO ARRAY [0..0] OF UDINT
END_METHOD

(* Returns the explicitely selected alarm groups. The array contains the internal IDs of the alarm groups to consider.*)
METHOD GetAlarmGroups : POINTER TO ARRAY [0..0] OF UDINT
GetAlarmGroups := pudiAlarmGroupIDs;
END_METHOD

{warning 'Add method implementation '}
(* Returns the number of explicitely selected alarm classes*)
METHOD GetCountAlarmClasses : INT
END_METHOD

(* Returns the number of explicitely selected alarm groups*)
METHOD GetCountAlarmGroups : INT
GetCountAlarmGroups := iCountAlarmGroups;
END_METHOD


(* Returns the lower bound of the priority filter range*)
METHOD GetPriorityFrom : USINT
GetPriorityFrom := 0;
END_METHOD

(* Returns the upper bound of the priority filter range*)
METHOD GetPriorityTo : USINT
GetPriorityTo := 255;
END_METHOD

END_FUNCTION_BLOCK

// Device/Application/Alarmy/ProcessAlarms
/// A function, that demonstrates, how to process the alarms, that we got from the alarm manager API.
/// This function prints the alarms to the console.
FUNCTION ProcessAlarms : BOOL
VAR_INPUT
	pitfAlarms	: POINTER TO ARRAY[0..0] OF IAlarm;
	udiCountAlarms: UDINT;
	
	pAlarmsAsString		: POINTER TO ARRAY[0..0] OF StructureAlarmAsStrings;
	udiCountAlarmsAsString: UDINT;
END_VAR
VAR
	i					: UDINT;
	itfAlarmGroup		: IAlarmGroup;
	itfAlarmClass		: IAlarmClass;
	liTimestamp			: AlarmManager.Timestamp;
	psMessage			: POINTER TO STRING;
	itfTypedValue		: ITypedValue;
	// Temporary string used to format timestamps
	dbsTempString		: Stu.CharBufferString(uiBufferSize := 200, stringType := __SYSTEM.TYPE_CLASS.TYPE_STRING);
	// We use this severity, so that the output will be visible on the console without modifying the
	// configuration file of the PLC
	udiSeverity			: UDINT := VisuElems.LogClass.LOG_ERROR;
	
	AlarmString	: StructureAlarmAsStrings;
END_VAR

//VisuElems.Visu_Output('----------', udiSeverity);
IF 0 <> udiCountAlarms THEN
	FOR i := 0 TO udiCountAlarms - 1 DO
		itfAlarmGroup := pitfAlarms^[i].GetAlarmGroup();
		itfAlarmClass := pitfAlarms^[i].GetAlarmClass();
	//	VisuElems.Visu_Output_2('  Alarm ', UDINT_TO_STRING(i), udiSeverity);
		
		// first fill the AlarmTableSimulationRow variable and then print the data to the console
		AlarmString.sState			:= GetAlarmStateString(pitfAlarms^[i].GetState());
		AlarmString.sID			:= UINT_TO_STRING(pitfAlarms^[i].GetID());
		AlarmString.sInternalID	:= UDINT_TO_STRING(pitfAlarms^[i].GetInternalID());
		IF 0 = itfAlarmGroup THEN
			// Might happen if in the alarm storage an old row was read, where the alarm group is
			// no longer valid
			AlarmString.sAlarmGroup	:= '???';
		ELSE	
			AlarmString.sAlarmGroup	:= itfAlarmGroup.GetName();
		END_IF
		
		liTimestamp := pitfAlarms^[i].GetTimestampLast();
		FormatTimestamp(liTimestamp, dbsTempString);
		AlarmString.sTSLast		:= dbsTempString.m_AsString^;
		
		itfTypedValue := pitfAlarms^[i].GetLatchVar1Value();
		FormatTypedValue(itfTypedValue, dbsTempString);
		AlarmString.sLatchVar1		:= dbsTempString.m_AsString^;
		
		itfTypedValue := pitfAlarms^[i].GetLatchVar2Value();
		FormatTypedValue(itfTypedValue, dbsTempString);
		AlarmString.sLatchVar2		:= dbsTempString.m_AsString^;

		itfTypedValue := pitfAlarms^[i].GetCurrentValue();
		FormatTypedValue(itfTypedValue, dbsTempString);
		AlarmString.sCurrValue		:= dbsTempString.m_AsString^;
		
		IF itfAlarmClass <> 0 THEN
			AlarmString.sAlarmClass	:= itfAlarmClass.GetName();
			AlarmString.sPriority		:= USINT_TO_STRING(itfAlarmClass.GetPriority());
		ELSE
			AlarmString.sAlarmClass	:= '???';
			AlarmString.sPriority		:= '???';
		END_IF


		IF 0 = itfAlarmGroup THEN
			// Might happen if in the alarm storage an old row was read, where the alarm group is
			// no longer valid
			AlarmString.sMessage	:= '???';
		ELSE	
			psMessage := pitfAlarms^[i].GetMessage(stringType := __SYSTEM.TYPE_CLASS.TYPE_STRING);
			AlarmString.sMessage		:= psMessage^;
		END_IF
(*		
		// Print data
		VisuElems.Visu_Output_2('    State      : ', AlarmString.sState,		udiSeverity);
		VisuElems.Visu_Output_2('    ID         : ', AlarmString.sID,			udiSeverity);
		VisuElems.Visu_Output_2('    internal ID: ', AlarmString.sInternalID,	udiSeverity);
		VisuElems.Visu_Output_2('    Alarm group: ', AlarmString.sAlarmGroup,	udiSeverity);
		VisuElems.Visu_Output_2('    TS last    : ', AlarmString.sTSLast,		udiSeverity);
		VisuElems.Visu_Output_2('    Message    : ', AlarmString.sMessage,		udiSeverity);
		VisuElems.Visu_Output_2('    CurrValue  : ', AlarmString.sCurrValue,	udiSeverity);
		VisuElems.Visu_Output_2('    LatchVar1  : ', AlarmString.sLatchVar1,	udiSeverity);
		VisuElems.Visu_Output_2('    LatchVar2  : ', AlarmString.sLatchVar2,	udiSeverity);
		VisuElems.Visu_Output_2('    Class      : ', AlarmString.sAlarmClass,	udiSeverity);
		VisuElems.Visu_Output_2('    Priority   : ', AlarmString.sPriority,	udiSeverity);
		VisuElems.Visu_Output('-------------------------------', udiSeverity);
*)		
		
		// If a valid pointer to an array has been passed, we also store it in the array
		IF pAlarmsAsString <> 0 AND i < udiCountAlarmsAsString THEN
			pAlarmsAsString^[i] := AlarmString;
		END_IF
		
	END_FOR
END_IF

//	VisuElems.Visu_Output('-------------------------------', udiSeverity);
// Necessary to free the memory, that was allocated by FB_Init
dbsTempString.FB_Exit(FALSE);

END_FUNCTION

// Device/Application/Obiekty/FB_Kolumna
FUNCTION_BLOCK FB_Kolumna IMPLEMENTS I_Kolumna
VAR_INPUT
END_VAR
VAR_OUTPUT
END_VAR
VAR
	fbImpulsator: BLINK;
	xEnableImpulsator: BOOL;
	fbTimerPrzerwa: TON;
	xEnableTimerPrzerwa: BOOL;
	tCzasPrzerwy: TIME;
	eKolor : (ZIELONY, CZERWONY, ZOLTY, NIEBIESKI);
END_VAR

fbImpulsator(ENABLE:= xEnableImpulsator, TIMELOW:= T#500MS, TIMEHIGH:= T#500MS );
fbTimerPrzerwa(IN:= xEnableTimerPrzerwa, PT:= T#1M, ET=> tCzasPrzerwy);

{warning 'Add method implementation '}
METHOD M_BuzzerOnOff : BOOL
VAR_INPUT
	in_xOnOff	: BOOL;
END_VAR
VAR_OUTPUT
	out_xBuzzer	: BOOL;
END_VAR
IF in_xOnOff THEN
	xEnableTimerPrzerwa := TRUE;
ELSE
	xEnableTimerPrzerwa := FALSE;
END_IF

out_xBuzzer := fbTimerPrzerwa.Q;
END_METHOD

{warning 'Add method implementation '}
METHOD M_UstawKolor : INT
VAR_INPUT
	in_xEnable	: BOOL;
	(* 0 - czerwony, 1 - zielony, 2 - żółty, 3 - niebieski*)
	in_iKolor	: INT;
	in_xImpusatorOnOff	: BOOL;
END_VAR
VAR_OUTPUT
	out_xZielony	: BOOL;
	out_xCzerwony	: BOOL;
	out_xZolty	: BOOL;
	out_xNiebieski	: BOOL;
END_VAR
xEnableImpulsator := in_xEnable;
IF in_xEnable THEN
	CASE in_iKolor OF
		ZIELONY:
				IF in_xImpusatorOnOff THEN
					out_xZielony := fbImpulsator.OUT;
				ELSE
					out_xZielony := TRUE;
				END_IF
		CZERWONY:
				IF in_xImpusatorOnOff THEN
					out_xCzerwony := fbImpulsator.OUT;
				ELSE
					out_xCzerwony := TRUE;
				END_IF
		ZOLTY:
				IF in_xImpusatorOnOff THEN
					out_xZolty := fbImpulsator.OUT;
				ELSE
					out_xZolty := TRUE;
				END_IF
		NIEBIESKI:
				IF in_xImpusatorOnOff THEN
					out_xNiebieski := fbImpulsator.OUT;
				ELSE
					out_xNiebieski := TRUE;
				END_IF
	END_CASE
ELSE
	out_xZielony := FALSE; out_xCzerwony := FALSE; out_xZolty := FALSE; out_xNiebieski := FALSE;
END_IF
END_METHOD

END_FUNCTION_BLOCK

// Device/Application/Interfejsy/I_Kolumna
INTERFACE I_Kolumna

METHOD M_BuzzerOnOff : BOOL
VAR_INPUT
	in_xOnOff: BOOL;
END_VAR

VAR_OUTPUT
	out_xBuzzer: BOOL;
END_VAR
END_METHOD

METHOD M_UstawKolor : INT
VAR_INPUT
	in_xEnable: BOOL;
	in_iKolor	: INT; // 0 - czerwony, 1 - zielony, 2 - żółty, 3 - niebieski
	in_xImpusatorOnOff: BOOL;
END_VAR

VAR_OUTPUT
	out_xZielony: BOOL;
	out_xCzerwony: BOOL;
	out_xZolty: BOOL;
	out_xNiebieski: BOOL;
END_VAR
END_METHOD

END_INTERFACE

// Device/Application/Programy/Sortery
PROGRAM Sortery
VAR
	Sorter1: Sorter_1;
	Sorter2: Sorter_1;
	Sorter3: Sorter_1;

	diNumerProduktuTemp:DINT;
	Predkosc: INT;
END_VAR

VAR RETAIN
      iIndeksSortera1 { S7_SetPoint := 'True'} : INT:=1;
      iIndeksSortera2 { S7_SetPoint := 'True'} : INT:=13;
      iIndeksSortera3 { S7_SetPoint := 'True'} : INT:=24;
 END_VAR

IF FIO.xFIOAktywny THEN

// podział parametryzacji sorterów w przypadku stanu startu i stopu linii
IF GVL.xLiniaStart OR PLC_PRG.fbPrzenosnik.Predkosc > 0 THEN // praca linii, sortowanie uruchomione
	// sorter 1, produkty zielone 4-6
	//
	Sorter1.in_xSortuj := 1;  // sortowanie
	Sorter1.in_xBazuj := 0;
	IF GVL.aRejestrProduktow[iIndeksSortera1] >= 4 AND GVL.aRejestrProduktow[iIndeksSortera1] <= 6 THEN
		Sorter1.in_xExecute := 1;
		GVL.aRejestrProduktow[iIndeksSortera1] := 0;
	ELSE
		Sorter1.in_xExecute := 0;
	END_IF;
	// sorter 2, produkty niebieskie 1-3
	//
	Sorter2.in_xSortuj := 1;  // sortowanie
	Sorter2.in_xBazuj := 0;
	IF GVL.aRejestrProduktow[iIndeksSortera2] >= 1 AND GVL.aRejestrProduktow[iIndeksSortera2] <= 3 THEN
		Sorter2.in_xExecute := 1;
		GVL.aRejestrProduktow[iIndeksSortera2] := 0;
	ELSE
		Sorter2.in_xExecute := 0;
	END_IF;
	// sorter 3, produkty szare 6-9
	//
	Sorter3.in_xSortuj := 1;  // sortowanie
	Sorter3.in_xBazuj := 0;
	IF GVL.aRejestrProduktow[iIndeksSortera3] >= 6 AND GVL.aRejestrProduktow[iIndeksSortera3] <= 9 THEN
		Sorter3.in_xExecute := 1;
		diNumerProduktuTemp:=GVL.aRejestrProduktow[iIndeksSortera3];
	   GVL.aRejestrProduktow[iIndeksSortera3] := 0;
	ELSE
		Sorter3.in_xExecute := 0;
	END_IF;
ELSE    // zatrzymanie linii, bazowanie podczas zatrzymania
	Sorter1.in_xBazuj := 1;
	Sorter1.in_xSortuj := 0;
	Sorter1.in_xExecute := GVL.R_TRIG_Reset.Q;
	Sorter2.in_xBazuj := 1;
	Sorter2.in_xSortuj := 0;
	Sorter2.in_xExecute := (* GVL.R_TRIG_Reset.Q *) fio.xPrzyciskReset;
	Sorter3.in_xBazuj := 1;
	Sorter3.in_xSortuj := 0;
	Sorter3.in_xExecute := GVL.R_TRIG_Reset.Q;
END_IF;

// wywołanie bloków funkcyjnych sorterów
Sorter1(in_xSensorZsuwni := fio.xCzujnikElementNOK_1,
		  in_xStartLinii :=GVL.xLiniaStart OR ( PLC_PRG.fbPrzenosnik.Predkosc > 0 ),
		  in_timWatchDogPT := T#2000ms,
		  out_xObrot => fio.xSorterObroc_1,
		  out_xPas => fio.xSorterPas_1);
Sorter2(in_xSensorZsuwni := fio.xCzujnikElementOK_2,
		  in_xStartLinii :=GVL.xLiniaStart OR ( PLC_PRG.fbPrzenosnik.Predkosc > 0 ),
		  in_timWatchDogPT := T#2000ms,
		  out_xObrot => fio.xSorterObroc_2,
		  out_xPas => fio.xSorterPas_2);
Sorter3(in_xSensorZsuwni := fio.xCzujnikElementOK_3,
		  in_xStartLinii :=GVL.xLiniaStart OR ( PLC_PRG.fbPrzenosnik.Predkosc > 0 ),
		  in_timWatchDogPT := T#2000ms,
		  out_xObrot => fio.xSorterObroc_3,
		  out_xPas => fio.xSorterPas_3);

GVL.R_TRIG_Start(CLK := fio.xPrzyciskStart);
GVL.R_TRIG_Reset(CLK := fio.xPrzyciskReset);

end_if;

END_PROGRAM

// Device/Application/Obiekty/Sorter
FUNCTION_BLOCK Sorter
 VAR_INPUT 
      in_xExecute : Bool;
      in_xSensorZsuwni : Bool;
      in_xSortuj : Bool;
      in_xBazuj : Bool;
      in_xStartLinii : Bool;
      in_timWatchDogPT : Time;
   END_VAR

   VAR_OUTPUT 
      out_xObrot : Bool;
      out_xPas : Bool;
      out_xDone : Bool;
      out_xBusy : Bool;
      out_xError : BOOL;
      out_wStatus : Word;
   END_VAR

   VAR 
      iKrok : Int;
      R_Trig_Start {InstructionName := 'R_TRIG'; LibVersion := '1.0'} : R_TRIG;
      Timer1 {InstructionName := 'TONR_TIME'; LibVersion := '1.0'} : TON;
      Timer2 {InstructionName := 'TON_TIME'; LibVersion := '1.0'} : TON;
      xTimer2_IN { S7_SetPoint := 'True'} : Bool;
      xTimer1_IN { S7_SetPoint := 'True'} : Bool;
      xTimer1_R : Bool;
      wErrorId : WORD;
	  eStanMaszyny: (INIT, SORTOWANIE, OCZEKIWANIE_NA_PRODUKT, SORTOWANIE_KONIEC, BAZOWANIE, BAZOWANIE_KONIEC, ERROR);
END_VAR


//=============================================================================
//ControlByte
//(c)Copyright (2020) All Rights Reserved
//-----------------------------------------------------------------------------
//Library:       Linia sortujaca
//Tested with:   S7 1200 4.2
//Engineering:   TIA Portal V15.1
//Restrictions:  -
//Requirements:  (hardware, technological package, memory needed, etc.)
//Functionality: Obsluga sortera
//-----------------------------------------------------------------------------
//Change log table:
//Version  Date       Expert in charge Changes applied
//01.00.00 02.10.2020 Kamil Biedulski First released version
//=============================================================================
//

R_Trig_Start(CLK:=in_xExecute);

Timer1(IN:=xTimer1_IN,
		//R:=xTimer1_R,
		PT:=in_timWatchDogPT);
Timer2(IN:=xTimer2_IN,
		PT:=T#2S);


IF R_Trig_Start.Q THEN
	eStanMaszyny := INIT;
	wErrorId := 0;
END_IF;

CASE eStanMaszyny OF
	INIT :  // Init
		
		// sterowanie sorterem
		out_xObrot := 0;
		out_xPas := 0;
		
		// zmienne statusowe bloku
		out_xDone := 0;
		out_xBusy := 0;
		out_xError := 0;
		
		IF wErrorId <> 0 THEN
			out_wStatus := wErrorId;
		ELSE
			out_wStatus := 16#7000;
		END_IF;
		
		xTimer1_IN := 0;
		xTimer1_R := 1;
		xTimer2_IN := 0;
		
		// warunek tranzycji
		IF R_Trig_Start.Q THEN

			IF in_xSortuj AND NOT in_xBazuj THEN
				iKrok := 10;
				out_wStatus := 16#7001;
				out_xObrot := 1;
				out_xPas := in_xStartLinii;
			ELSIF in_xBazuj AND NOT in_xSortuj THEN
				iKrok := 30;
				out_wStatus := 16#7001;
			END_IF;
			
			IF NOT (in_xSortuj XOR in_xBazuj) THEN
				wErrorId := 16#8200;
				iKrok := 100;
			END_IF;

		END_IF;
		
		IF NOT in_xSensorZsuwni THEN
			wErrorId := 16#8202;
			iKrok := 100;
		END_IF;
		
	SORTOWANIE:  // Cykl sortowania
		
		// sterowanie sorterem
		out_xObrot := 1;
		out_xPas := in_xStartLinii;
		
		// zmienne statusowe bloku
		out_xDone := 0;
		out_xBusy := 1;
		out_xError := 0;
		
		out_wStatus := 16#7002;
		
		// timer
		xTimer1_IN := in_xStartLinii;
		xTimer1_R := 0;
		
		// warunek tranzycji
		IF NOT in_xSensorZsuwni THEN
			iKrok := 15;
		ELSIF Timer1.Q THEN
			wErrorId := 16#8201;
			iKrok := 100;
		END_IF;
		
	OCZEKIWANIE_NA_PRODUKT: // Oczekiwanie na zsunięcie produktu
			
			// sterowanie sorterem
			out_xObrot := 1;
			out_xPas := in_xStartLinii;
			
			// zmienne statusowe bloku
			out_xDone := 0;
			out_xBusy := 1;
			out_xError := 0;
			
			out_wStatus := 16#7002;
			
			// timer
			xTimer1_IN := in_xStartLinii;
			xTimer1_R := 0;
			
			// warunek tranzycji
			IF in_xSensorZsuwni THEN
				iKrok := 20;
			ELSIF Timer1.Q THEN
				wErrorId := 16#8201;
				iKrok := 100;
			END_IF;
		
	SORTOWANIE_KONIEC: // Koniec cyklu sortowania
		
		// sterowanie sorterem
		out_xObrot := 0;
		out_xPas := 0;
		
		// zmienne statusowe bloku
		out_xDone := 1;
		out_xBusy := 0;
		out_xError := 0;
		
		out_wStatus := 16#0000;
		
		// warunek tranzycji
		IF NOT in_xExecute THEN
			iKrok := 0;
		END_IF;
	BAZOWANIE:  // Cykl bazowania
		
		// sterowanie sorterem
		out_xObrot := 0;
		out_xPas := 0;
		
		// zmienne statusowe bloku
		out_xDone := 0;
		out_xBusy := 1;
		out_xError := 0;
		
		out_wStatus := 16#7002;
		
		// timer
		xTimer2_IN := 1;
		
		// warunek tranzycji
		IF Timer2.Q THEN
			iKrok := 40;
		END_IF;
		
	BAZOWANIE_KONIEC: // Koniec cyklu bazowania
		
		// sterowanie sorterem
		out_xObrot := 0;
		out_xPas := 0;
		
		// zmienne statusowe bloku
		out_xDone := 1;
		out_xBusy := 0;
		out_xError := 0;
		
		out_wStatus := 16#0000;
		
		// warunek tranzycji
		IF NOT in_xExecute THEN
			iKrok := 0;
		END_IF;
		
	ERROR:    // Obsługa błędów
		
		// sterowanie sorterem
	  //  out_xObrot := 0;
		out_xPas := 0;
		
		// zmienne statusowe bloku
		out_xDone := 0;
		out_xBusy := 0;
		out_xError := 1;
		
		out_wStatus := wErrorId;
		
		// warunek tranzycji
		IF NOT in_xExecute THEN
			iKrok := 0;
		END_IF;
		
	ELSE  // Statement section ELSE
		;
END_CASE;

END_FUNCTION_BLOCK

// Device/Application/Obiekty/Sorter_1
FUNCTION_BLOCK Sorter_1
 VAR_INPUT 
      in_xExecute : Bool;
      in_xSensorZsuwni : Bool;
      in_xSortuj : Bool;
      in_xBazuj : Bool;
      in_xStartLinii : Bool;
      in_timWatchDogPT : Time;
   END_VAR

   VAR_OUTPUT 
      out_xObrot : Bool;
      out_xPas : Bool;
      out_xDone : Bool;
      out_xBusy : Bool;
      out_xError : Bool;
      out_wStatus : Word;
   END_VAR

   VAR 
      iKrok : Int;
      R_Trig_Start {InstructionName := 'R_TRIG'; LibVersion := '1.0'} : R_TRIG;
      Timer1 {InstructionName := 'TONR_TIME'; LibVersion := '1.0'} : TON;
      Timer2 {InstructionName := 'TON_TIME'; LibVersion := '1.0'} : TON;
      xTimer2_IN { S7_SetPoint := 'True'} : Bool;
      xTimer1_IN { S7_SetPoint := 'True'} : Bool;
      xTimer1_R : Bool;
      wErrorId : WORD;
	  eStanMaszyny: (INIT, SORTOWANIE, OCZEKIWANIE_NA_PRODUKT, SORTOWANIE_KONIEC, BAZOWANIE_SORTERA, BAZOWANIE_KONIEC, ERROR);
END_VAR


//=============================================================================
//ControlByte
//(c)Copyright (2020) All Rights Reserved
//-----------------------------------------------------------------------------
//Library:       Linia sortujaca
//Tested with:   S7 1200 4.2
//Engineering:   TIA Portal V15.1
//Restrictions:  -
//Requirements:  (hardware, technological package, memory needed, etc.)
//Functionality: Obsluga sortera
//-----------------------------------------------------------------------------
//Change log table:
//Version  Date       Expert in charge Changes applied
//01.00.00 02.10.2020 Kamil Biedulski First released version
//=============================================================================
//

R_Trig_Start(CLK:=in_xExecute);

Timer1(IN:=xTimer1_IN,
		//R:=xTimer1_R,
		PT:=in_timWatchDogPT);
Timer2(IN:=xTimer2_IN,
		PT:=T#2S);


IF R_Trig_Start.Q THEN
	eStanMaszyny := INIT;
	wErrorId := 0;
END_IF;

CASE eStanMaszyny OF
	INIT: 
		Init();
		TRANS_INIT;
		
	SORTOWANIE:
		Sortowanie();
		TRANS_SORTOWANIE;
		
	OCZEKIWANIE_NA_PRODUKT:
		Czekaj();
		TRANS_CZEKAJ;
	
	SORTOWANIE_KONIEC:
		SortowanieKoniec();
		TRANS_SORTOWANIE_KONIEC;
	
	
	BAZOWANIE_SORTERA:
		Bazowanie();
		TRANS_BAZOWANIE;
	
	BAZOWANIE_KONIEC:
		Bazowanie_koniec();
		TRANS_BAZOWANIE_KONIEC;
	ERROR:
		Error();
		TRANS_ERROR;
		
		
		
		
END_CASE

METHOD PRIVATE Bazowanie : BOOL
VAR_INPUT
END_VAR
// sterowanie sorterem
out_xObrot := 0;
out_xPas := 0;

// zmienne statusowe bloku
out_xDone := 0;
out_xBusy := 1;
out_xError := 0;

out_wStatus := 16#7002;

// timer
xTimer2_IN := 1;
END_METHOD

METHOD PRIVATE Bazowanie_koniec : BOOL
VAR_INPUT
END_VAR
// sterowanie sorterem
out_xObrot := 0;
out_xPas := 0;

// zmienne statusowe bloku
out_xDone := 1;
out_xBusy := 0;
out_xError := 0;

out_wStatus := 16#0000;
END_METHOD

METHOD PRIVATE Czekaj : BOOL
VAR_INPUT
END_VAR
// sterowanie sorterem
out_xObrot := 1;
out_xPas := in_xStartLinii;

// zmienne statusowe bloku
out_xDone := 0;
out_xBusy := 1;
out_xError := 0;

out_wStatus := 16#7002;

// timer
xTimer1_IN := in_xStartLinii;
xTimer1_R := 0;
END_METHOD

METHOD PRIVATE Error : BOOL
VAR_INPUT
END_VAR
// sterowanie sorterem
//  out_xObrot := 0;
out_xPas := 0;

// zmienne statusowe bloku
out_xDone := 0;
out_xBusy := 0;
out_xError := 1;

out_wStatus := wErrorId;
END_METHOD

//FB_Init is always available implicitly and it is used primarily for initialization.
//The return value is not evaluated. For a specific influence, you can also declare the
//methods explicitly and provide additional code there with the standard initialization
//code. You can evaluate the return value.
METHOD FB_Init: BOOL
VAR_INPUT
    bInitRetains: BOOL; // TRUE: the retain variables are initialized (reset warm / reset cold)
    bInCopyCode: BOOL;  // TRUE: the instance will be copied to the copy code afterward (online change)   
END_VAR

		out_xObrot := 0;
		out_xPas := 0;
		
		// zmienne statusowe bloku
		out_xDone := 0;
		out_xBusy := 0;
		out_xError := 0;
		
		IF wErrorId <> 0 THEN
			out_wStatus := wErrorId;
		ELSE
			out_wStatus := 16#7000;
		END_IF;
		
		xTimer1_IN := 0;
		xTimer1_R := 1;
		xTimer2_IN := 0;
END_METHOD

METHOD PRIVATE Init : bool
VAR_INPUT
END_VAR
out_xObrot := 0;
out_xPas := 0;

// zmienne statusowe bloku
out_xDone := 0;
out_xBusy := 0;
out_xError := 0;

IF wErrorId <> 0 THEN
	out_wStatus := wErrorId;
ELSE
	out_wStatus := 16#7000;
END_IF;

xTimer1_IN := 0;
xTimer1_R := 1;
xTimer2_IN := 0;
END_METHOD

METHOD PRIVATE Sortowanie : BOOL
VAR_INPUT
END_VAR
// sterowanie sorterem
out_xObrot := 1;
out_xPas := in_xStartLinii;

// zmienne statusowe bloku
out_xDone := 0;
out_xBusy := 1;
out_xError := 0;

out_wStatus := 16#7002;

// timer
xTimer1_IN := in_xStartLinii;
xTimer1_R := 0;
END_METHOD

METHOD PRIVATE SortowanieKoniec : BOOL
VAR_INPUT
END_VAR
// sterowanie sorterem
out_xObrot := 0;
out_xPas := 0;

// zmienne statusowe bloku
out_xDone := 1;
out_xBusy := 0;
out_xError := 0;

out_wStatus := 16#0000;
END_METHOD

TRANSITION TRANS_BAZOWANIE:
// warunek tranzycji
IF Timer2.Q THEN
	eStanMaszyny := BAZOWANIE_KONIEC;
END_IF;
END_TRANSITION

TRANSITION TRANS_BAZOWANIE_KONIEC:
	// warunek tranzycji
	IF NOT in_xExecute THEN
		eStanMaszyny := INIT;
	END_IF;
END_TRANSITION

TRANSITION TRANS_CZEKAJ:
// warunek tranzycji
IF in_xSensorZsuwni THEN
	eStanMaszyny := SORTOWANIE_KONIEC;
ELSIF Timer1.Q THEN
	wErrorId := 16#8201;
	eStanMaszyny := ERROR;
END_IF;
END_TRANSITION

TRANSITION TRANS_ERROR:
// warunek tranzycji
IF NOT in_xExecute THEN
	eStanMaszyny := INIT;
END_IF;
END_TRANSITION

TRANSITION TRANS_INIT:
// warunek tranzycji
IF R_Trig_Start.Q THEN

	IF in_xSortuj AND NOT in_xBazuj THEN
		eStanMaszyny := SORTOWANIE;
		out_wStatus := 16#7001;
		out_xObrot := 1;
		out_xPas := in_xStartLinii;
	ELSIF in_xBazuj AND NOT in_xSortuj THEN
		eStanMaszyny := SORTOWANIE_KONIEC;
		out_wStatus := 16#7001;
	END_IF;
	
	IF NOT (in_xSortuj XOR in_xBazuj) THEN
		wErrorId := 16#8200;
		eStanMaszyny := ERROR;
	END_IF;

END_IF;

IF NOT in_xSensorZsuwni THEN
	wErrorId := 16#8202;
	eStanMaszyny := ERROR;
END_IF;
END_TRANSITION

TRANSITION TRANS_SORTOWANIE:
// warunek tranzycji
IF NOT in_xSensorZsuwni THEN
	eStanMaszyny := OCZEKIWANIE_NA_PRODUKT;
ELSIF Timer1.Q THEN
	wErrorId := 16#8201;
	eStanMaszyny := ERROR;
END_IF;
END_TRANSITION

TRANSITION TRANS_SORTOWANIE_KONIEC:
// warunek tranzycji
IF NOT in_xExecute THEN
	eStanMaszyny := INIT;
END_IF;
END_TRANSITION

END_FUNCTION_BLOCK

// Device/Application/Programy/LogowanieDanych
PROGRAM LogowanieDanych
VAR
	eEventType1 : E_EventType := E_EventType.Alarm;
	eEventSeverity1: E_EventSeverity := E_EventSeverity.Error;
	nEventIdentity1 : UDINT := 42;
	sEventText1 : STRING(255) := 'To jest poważny alarm';
	
	
	CsvPersistentEventStorage : FB_CsvPersistentEventStorage;
	EventLogger: FB_EventLogger(CsvPersistentEventStorage) ;
	
	xBool:BOOL ;
	
	xInit	: BOOL;
	udiCreateError: UDINT;
	
	Impulsator: BLINK;
	rtrig1: R_TRIG;
	
	fbXmlPac: FB_XmlPac;
	EventLoggerXml: FB_EventLogger(fbXmlPac) ;
	fbRtrigEstop: r_trig;
	fbRtrigHold: r_trig;
	fbRtrigSuspended: r_trig;
END_VAR

fbRtrigEstop(CLK := NOT fio.xEmergencyStop );
fbRtrigHold(CLK := PLC_PRG.xHold );
fbRtrigSuspended(CLK :=  PLC_PRG.xSuspend );
IF fbRtrigEstop.Q THEN
	eEventType1 := E_EventType.Alarm;
	eEventSeverity1 := E_EventSeverity.Critical;
	nEventIdentity1 := 1;
	sEventText1 := 'Emergency Stop';
	EventLogger.AddEvent(eEventType1, eEventSeverity1, nEventIdentity1, sEventText1);	
END_IF

IF fbRtrigHold.Q THEN
	eEventType1 := E_EventType.Message;
	eEventSeverity1 := E_EventSeverity.Info;
	nEventIdentity1 := 2;
	sEventText1 := 'Maszyna w stanie HELD';
	EventLogger.AddEvent(eEventType1, eEventSeverity1, nEventIdentity1, sEventText1);
END_IF

IF fbRtrigSuspended.Q THEN
	eEventType1 := E_EventType.Message;
	eEventSeverity1 := E_EventSeverity.Warning;
	nEventIdentity1 := 3;
	sEventText1 := 'Maszyna w stanie SUSPENDED';
	EventLogger.AddEvent(eEventType1, eEventSeverity1, nEventIdentity1, sEventText1);
END_IF


CsvPersistentEventStorage();

END_PROGRAM

// Device/Application/Data logger/FB_CsvPersistentEventStorage
FUNCTION_BLOCK FB_CsvPersistentEventStorage IMPLEMENTS I_PersistentEventStorage
VAR_INPUT
END_VAR
VAR_OUTPUT
END_VAR
VAR
	
	sFileName 		: CAA.FILENAME;
	sFileNameCopy 	: CAA.FILENAME;	
	fbFileOpen 		: File.Open := (eFileMode:= File.MODE.MWRITE OR File.MODE.MAPPD) ;
	fbFileClose		: File.Close;
	FileCopy		: File.Copy;
	GetFileSize		: File.GetSize;
	GetFileTime		: File.GetTime;
	FileRead		: File.Read;
	fbFileWrite		: File.Write;
	SetFilePos		: File.SetPos;
	GetFilePos		: File.GetPos;	
	iState			: UINT;	
	hfile			: CAA.HANDLE;
	sWriteLine		: STRING(128);
	sReadLine		: STRING;	
	dtModification 	: DATE_AND_TIME;
	udiFileSize		: __XWORD;
	xError			: BOOL := FALSE;
	xInit			: BOOL := FALSE;
	xTestDone		: BOOL := FALSE;
	xStartTest		: BOOL := TRUE; 

	eWriteState : (FILE_OPEN_TRIGGER, FILE_OPEN, WAIT_FOR_EVENT, WRITE_EVENT_TRIGGER, WRITE_EVENT, FILE_CLOSE_TRIGGER, FILE_CLOSE, FILE_OPEN_READ, ERROR);
	stEventWrittenToFile: ST_Event; 	
	CsvString: STRING(E_MaxString.MaxString);
END_VAR

IF xStartTest THEN
	sFileName := '/testcodesys.txt';
	sFileName := CONCAT(gvl.g_sMainDirectory, sFileName);
	sFileNameCopy := '/CAAFileCopy.txt';
	sFileNameCopy := CONCAT(gvl.g_sMainDirectory, sFileNameCopy);
	//eWriteState := FILE_OPEN_TRIGGER;
	xTestDone := FALSE;
	xError := FALSE;
	xStartTest := FALSE;
END_IF

 CASE eWriteState OF
	 FILE_OPEN_TRIGGER:
	 	fbFileOpen(xExecute := TRUE,sFileName:= sFileName, xExclusive:= FALSE, eFileMode:= File.MODE.MWRITE ); (* OR File.MODE.MAPPD) *)
		eWriteState := FILE_OPEN;
	 FILE_OPEN:
	   fbFileOpen(xExecute:= FALSE);
	   IF NOT fbFileOpen.xBusy (* AND fbFileOpen.hFile <> 0 *) THEN		   
		   hfile := fbFileOpen.hFile;		   
		   eWriteState := WAIT_FOR_EVENT;
	   ELSIF fbFileOpen.xError = TRUE THEN
		   eWriteState := ERROR;
		   fbFileOpen(xExecute:= FALSE);
	   END_IF
	 WAIT_FOR_EVENT:
	 		// DO NOTHING
	 WRITE_EVENT_TRIGGER:
	 		CsvString := CreateCsvString(stEvent := stEventWrittenToFile);
	 		fbFileWrite(xExecute := TRUE, hFile := hfile, pBuffer:= ADR(CsvString), szSize:= INT_TO_UDINT(LEN(CsvString)));
			eWriteState := WRITE_EVENT;
	 WRITE_EVENT:
	 		fbFileWrite(xExecute:= FALSE);
	 	   IF NOT fbFileWrite.xBusy THEN			   
			   eWriteState := FILE_CLOSE_TRIGGER;
	  	   ELSIF fbFileWrite.xError = TRUE THEN			   
			   fbFileWrite(xExecute:= FALSE);
			   eWriteState:= ERROR;
	       END_IF
	 FILE_CLOSE_TRIGGER:
	 		fbFileClose(xExecute := TRUE, hFile := hfile);
	 		eWriteState := FILE_CLOSE;
	 FILE_CLOSE:
	 		fbFileClose(xExecute := FALSE);
			IF NOT fbFileClose.xBusy THEN
				eWriteState := FILE_OPEN_READ;
	 		ELSIF fbFileClose.xError THEN
				fbFileClose(xExecute := FALSE);
				eWriteState := ERROR;
			END_IF
	FILE_OPEN_READ: // Open the file again, with read append access.
	  fbFileOpen(xExecute := TRUE, sFileName:= sFileName, xExclusive:= FALSE, eFileMode:= File.MODE.MAPPD );
	  IF NOT fbFileOpen.xBusy (* AND fbFileOpen.hFile <> 0 *) THEN		   
		   hfile := fbFileOpen.hFile;		   
		   eWriteState := WAIT_FOR_EVENT;
		   fbFileOpen(xExecute := FALSE);
	  ELSIF fbFileOpen.xError = TRUE THEN
		   eWriteState := ERROR;
		   fbFileOpen(xExecute:= FALSE);
	  END_IF
	
	ERROR: 
	 
	 	// DO NOTHING 
 END_CASE

METHOD PRIVATE CreateCsvString : STRING(E_MaxString.MaxString)
VAR_INPUT
	stEvent : REFERENCE TO ST_Event;
END_VAR
VAR
	TempString: STRING(E_MaxString.MaxString);
END_VAR
TempString := TO_STRING(stEvent.eEventType);
TempString := CONCAT(STR1:= TempString, STR2:= ',');
TempString := CONCAT(STR1:= TempString, STR2:= TO_STRING(stEvent.eEventSeverity));
TempString := CONCAT(STR1:= TempString, STR2:= ',');
TempString := CONCAT(STR1 := TempString, STR2 := TO_STRING(stEvent.nEventIdentity));
TempString := CONCAT(STR1 := TempString, STR2 := ',');
TempString := CONCAT(STR1 := TempString, STR2 := stEvent.sEventText );
TempString := CONCAT(STR1 := TempString, STR2 := ',');
TempString := CONCAT(STR1 := TempString, STR2 := TO_STRING(stEvent.dtTimeStamp));
TempString := CONCAT(STR1 := TempString, STR2 := '$n');

CreateCsvString := TempString;
END_METHOD

{warning 'Add method implementation '}
METHOD StoreEvent
VAR_INPUT
	stEvent	: ST_Event;
END_VAR
IF eWriteState = WAIT_FOR_EVENT THEN
	eWriteState := WRITE_EVENT_TRIGGER;
	stEventWrittenToFile := stEvent;
END_IF
END_METHOD

END_FUNCTION_BLOCK

// Device/Application/Interfejsy/I_PersistentEventStorage
INTERFACE I_PersistentEventStorage

METHOD StoreEvent
VAR_INPUT
	stEvent: ST_Event;
END_VAR
END_METHOD

END_INTERFACE

// Device/Application/Data logger/FB_EventLogger
FUNCTION_BLOCK FB_EventLogger
VAR
	aEventBuffer: ARRAY[1..100] OF ST_Event; 
	CurrentEventBUfferIndex: INT := 0;
	
	_PersistentEventStorage : I_PersistentEventStorage;
END_VAR
VAR CONSTANT
	MAXIMUM_SIZE_OF_EVENT_BUFFER: INT := 100;
END_VAR

METHOD PUBLIC AddEvent : BOOL
VAR_INPUT
	eEventType : E_EventType;
	eEventSeverity: E_EventSeverity;
	nEventIdentity : UDINT;
	sEventText : STRING(255);
END_VAR
 IF NOT IsEventBufferFull() THEN
	CurrentEventBUfferIndex := CurrentEventBUfferIndex + 1;
	aEventBuffer[CurrentEventBufferIndex].eEventType := eEventType;
	aEventBuffer[CurrentEventBufferIndex].eEventSeverity := eEventSeverity;
	aEventBuffer[CurrentEventBufferIndex].nEventIdentity := nEventIdentity;
	aEventBuffer[CurrentEventBufferIndex].sEventText := sEventText;
	UpdateEventTimestampWithSystemTime(stEvent := aEventBuffer[CurrentEventBufferIndex]);
	AddEvent := TRUE;
ELSE
	AddEvent := FALSE;
END_IF

// mechanizm wstrzykiwania zależności
_PersistentEventStorage.StoreEvent(stEvent := aEventBuffer[CurrentEventBufferIndex]);
END_METHOD

//FB_Init is always available implicitly and it is used primarily for initialization.
//The return value is not evaluated. For a specific influence, you can also declare the
//methods explicitly and provide additional code there with the standard initialization
//code. You can evaluate the return value.
METHOD FB_Init: BOOL
VAR_INPUT
    bInitRetains: BOOL; // TRUE: the retain variables are initialized (reset warm / reset cold)
    bInCopyCode: BOOL;  // TRUE: the instance will be copied to the copy code afterward (online change)   
	iPersisentEventStorage : I_PersistentEventStorage;
END_VAR
_PersistentEventStorage := iPersisentEventStorage;
END_METHOD

METHOD PRIVATE IsEventBufferFull : BOOL
VAR_INPUT
END_VAR
IF (CurrentEventBUfferIndex + 1) > MAXIMUM_SIZE_OF_EVENT_BUFFER THEN
	IsEventBufferFull := TRUE;
ELSE
	IsEventBufferFull := FALSE;
END_IF
END_METHOD

END_FUNCTION_BLOCK

// Device/Application/Czas/UpdateEventTimestampWithSystemTime
FUNCTION UpdateEventTimestampWithSystemTime 
VAR_INPUT
	stEvent: REFERENCE TO ST_Event;
END_VAR
VAR
// 	fbGETSYSTEMTIME : GETSYSTEMTIME;	
// 	stFileTime : T_FILETIME;
END_VAR

// fbGETSYSTEMTIME(timeLoDW => stFileTime.dwHighDateTime,
// 				timeHiDW => stFileTime.dwHighDateTime);
				
stEvent.dtTimeStamp := PobranieCzasu();

END_FUNCTION

// Device/Application/Czas/PobranieCzasu
FUNCTION PobranieCzasu : DATE_AND_TIME
VAR_INPUT
END_VAR
VAR
	udiUtcTime 			: UDINT;
	udiUtcTimeLocal 	: UDINT;
	udiResult 			: UDINT;
	
	udiUTC_DateAndTime : UDINT;
    udiLocal_DateAndTime : UDINT;

    Result : SysTimeRtc.RTS_IEC_RESULT;
	

	dtNow: DATE_AND_TIME;
    todNow : TIME_OF_DAY; 
    datNow : DATE; 
END_VAR

// pobranie czasu UTC ze sterownika
udiUtcTime := SysTimeRtcGet(udiResult);
// konwersja czasu UTC do czasu lokalnego
udiResult := SysTimeRtcConvertUtcToLocal(udiUtcTime, udiUtcTimeLocal);
// konwersja czasu lokalnego do formatu Date_and_time
PobranieCzasu := UDINT_TO_DT(udiUtcTimeLocal);

dtNow := TO_DT(udiUtcTimeLocal); // DT#2018-6-6-9:8:38
todNow := TO_TOD(dtNow); // TOD#9:8:38
datNow := TO_DATE(dtNow); // D#2018-6-6

END_FUNCTION

// Device/Application/Data logger/FB_XmlPac
(*
    Demonstrates Xml parsing and composing
*)
FUNCTION_BLOCK FB_XmlPac IMPLEMENTS I_PersistentEventStorage
VAR
    xBufferInitialised : BOOL := FALSE;
	File : FB_FileControl;
	stFileAccessMode : SysFile.ACCESS_MODE := SysFile.AM_WRITE_PLUS;
	szFilename : STRING := 'C:\Temp\output.xml';
	
	Xml : FB_XmlControl;
	// select your buffertype
    Buffer : ARRAY [0..xmlpac.GVL_Param_XmlControl.MaxFileSize-1] OF BYTE;
    // or this buffertype
	////Buffer : STRING(GVL_Param_XmlControl.MaxFileSize);
	aEventBuffer: ARRAY[1..100] OF ST_Event; 
	CurrentEventBUfferIndex: INT := 0;
	
    xCreate : BOOL := TRUE ;
    xParse : BOOL := FALSE; 

    Status : SysFile.SysTypes.RTS_IEC_RESULT;
    result : xmlpac.E_XmlError;
    uiParseStep : DINT := 0;
	xRead : BOOL;
    XmlFileBytesRead : __XWORD;

    i : UINT;
    sTag : STRING;
	sPara : STRING;
	sTagPara : STRING;
    
    asParsedParameter1 : ARRAY[0..7] OF STRING;
    asParsedParameter2 : ARRAY[0..7] OF STRING;
    asParsedData : ARRAY[0..7] OF STRING;
    index : USINT := 0;
END_VAR

IF xCreate THEN
	//StoreEvent(stEvent := aEventBuffer[CurrentEventBUfferIndex]);
	xCreate := FALSE;
END_IF;

IF xParse THEN
	
    Parse();
END_IF

(*
    Creates an xml file
*)
METHOD ComposeXmlExample : BOOL
VAR_INPUT
END_VAR
Xml.writeDocumentHeader(Header := '<?xml version="1.0" encoding="UTF-8"?>');
Xml.newTag('users');
Xml.newTag('user');
Xml.NewParameter('age', '100');
Xml.NewParameter('sex', 'male');
Xml.newTagData('John Doe');
Xml.closeTag();
Xml.newTag('user');
Xml.NewParameter('age', '39');
Xml.NewParameter('sex', 'female');
Xml.newTagData('Jane Doe');
Xml.closeTag();
Xml.closeTag();

OpenWriteClose();
END_METHOD

METHOD FB_Init : BOOL
VAR_INPUT
  bInitRetains : BOOL; // TRUE: the retain variables are initialized (reset warm / reset cold)
  bInCopyCode : BOOL;  // TRUE: the instance will be copied to the copy code afterward (online change)
END_VAR
Xml.SetBuffer(pString := ADR(Buffer), iSizeOf := SIZEOF(Buffer));
xBufferInitialised := TRUE;
END_METHOD

METHOD OpenWriteClose : BOOL
VAR_INPUT
END_VAR
// write buffer to a file
File.Open(Filename := szFilename, FileAccessMode := stFileAccessMode);
File.Write(pString := ADR(Buffer), xml.Length );

File.Close();

Xml.ClearBuffer();
END_METHOD

ACTION Parse:
CASE uiParseStep OF
	0:  (* open file from start and read into buffer *)
        (* buffer is already set in FB_Init *)
		result := Xml.ReadFile(sFileName := szFilename, udiNextOffset := 0, BytesRead => XmlFileBytesRead);
		IF result = E_XmlError.Ok THEN
            index := 0;
            uiParseStep := 10;
        ELSE
            uiParseStep := 99;
        END_IF
        
	
	10:	(* the buffer is now filled in memory and the original file has been closed.
            So we can iterate it 
        *)
		sTag := Xml.NextTag();
        IF XML.sTagsSeek = '/users/user' THEN
            XML.NextParameter(Parameter => asParsedParameter1[index]);
            XML.NextParameter(Parameter => asParsedParameter2[index]);
            asParsedData[index] := XML.GetTagData();
            index := index + 1;
        ELSIF sTag = '/users' THEN
            // done
            uiParseStep := 100;
		ELSIF XML.SearchPos >= XML.Length THEN
			uiParseStep := 100 ;
		END_IF  
	
    99: (* error occured *)
        ;
        
	100:(* File does not contain usertags anymore *)
        ;
END_CASE
END_ACTION

{warning 'Add method implementation '}
METHOD StoreEvent
VAR_INPUT
	stEvent	: ST_Event;
// 	eEventType : E_EventType;
// 	eEventSeverity: E_EventSeverity;
// 	nEventIdentity : UDINT;
// 	sEventText : STRING(255);
// 	dtTimeStamp: DATE_AND_TIME;
END_VAR
// Xml.writeDocumentHeader(Header := '<?xml version="1.0" encoding="UTF-8"?>');
// Xml.newTag('users');
// Xml.newTag('Event Type');
// Xml.NewParameter('Severity', to_string(stEvent.eEventSeverity));
// Xml.NewParameter('sex', 'male');
// Xml.newTagData(TO_STRING(stEvent.eEventType));
// Xml.closeTag();
// Xml.newTag('user');
// Xml.NewParameter('age', '39');
// Xml.NewParameter('sex', 'female');
// Xml.newTagData('Jane Doe');
// Xml.closeTag();
// Xml.closeTag();
// 
// OpenWriteClose();

Xml.writeDocumentHeader(Header := '<?xml version="1.0" encoding="UTF-8"?>');
Xml.newTag('users');
Xml.newTag('Tekst');
Xml.NewParameter('Waznosc', TO_STRING(stEvent.eEventSeverity));
Xml.NewParameter('Typ',  TO_STRING(stEvent.eEventType));
Xml.newTagData(stEvent.sEventText);
Xml.closeTag();
Xml.newTag('Tekst');
Xml.NewParameter('Waznosc', TO_STRING(stEvent.eEventSeverity));
Xml.NewParameter('Typ',  TO_STRING(stEvent.eEventType));
Xml.newTagData(stEvent.sEventText);
Xml.closeTag();
Xml.closeTag();

OpenWriteClose();
END_METHOD

END_FUNCTION_BLOCK

// Device/Application/Programy/POU_cyclic
PROGRAM POU_cyclic
VAR
	iLicznik:INT;
	
	Impulsator: BLINK;
	rtrig1: R_TRIG;
	
	timInterwal: time;

END_VAR

// fio.iCzujnikWizyjny;

// logowanie danych co 1s
IF FIO.iPodajnikWyjsciowy > 0 THEN
timInterwal:=REAL_TO_TIME(360/FIO.iPodajnikWyjsciowy)/2;
ELSE
	timInterwal:=T#200MS;
END_IF;

Impulsator(ENABLE:= TRUE, TIMELOW:=timInterwal , TIMEHIGH:= timInterwal, OUT=> );
rtrig1(CLK:= Impulsator.OUT, Q=> );

IF ( GVL.xLiniaStart OR PLC_PRG.fbPrzenosnik.Predkosc > 0 ) AND rtrig1.q  THEN
    // przesunięcie elementów tablicy o jeden
    FOR iLicznik := 100 TO 1 BY -1 DO
        GVL.aRejestrProduktow[iLicznik] := GVL.aRejestrProduktow[iLicznik - 1];
    END_FOR;
    // wykrycie nowego produktu i wpisanie jego wartości do tablicy
    IF fio.iCzujnikWizyjny <> 0 AND fio.iCzujnikWizyjny  <> GVL.diSensorWizyjnyOstatniaWartosc THEN
        GVL.aRejestrProduktow[0] := fio.iCzujnikWizyjny ;
    ELSE
       GVL.aRejestrProduktow[0] := 0;
    END_IF;
    GVL.diSensorWizyjnyOstatniaWartosc := fio.iCzujnikWizyjny ;
ELSIF fio.xPrzyciskReset THEN
    // inicjalizacja wartości w tablicy
    FOR iLicznik := 0 TO 100 DO
        GVL.aRejestrProduktow[iLicznik] := 0;
    END_FOR;
   GVL.diSensorWizyjnyOstatniaWartosc := 0;
END_IF;

END_PROGRAM

// Device/Application/Panel
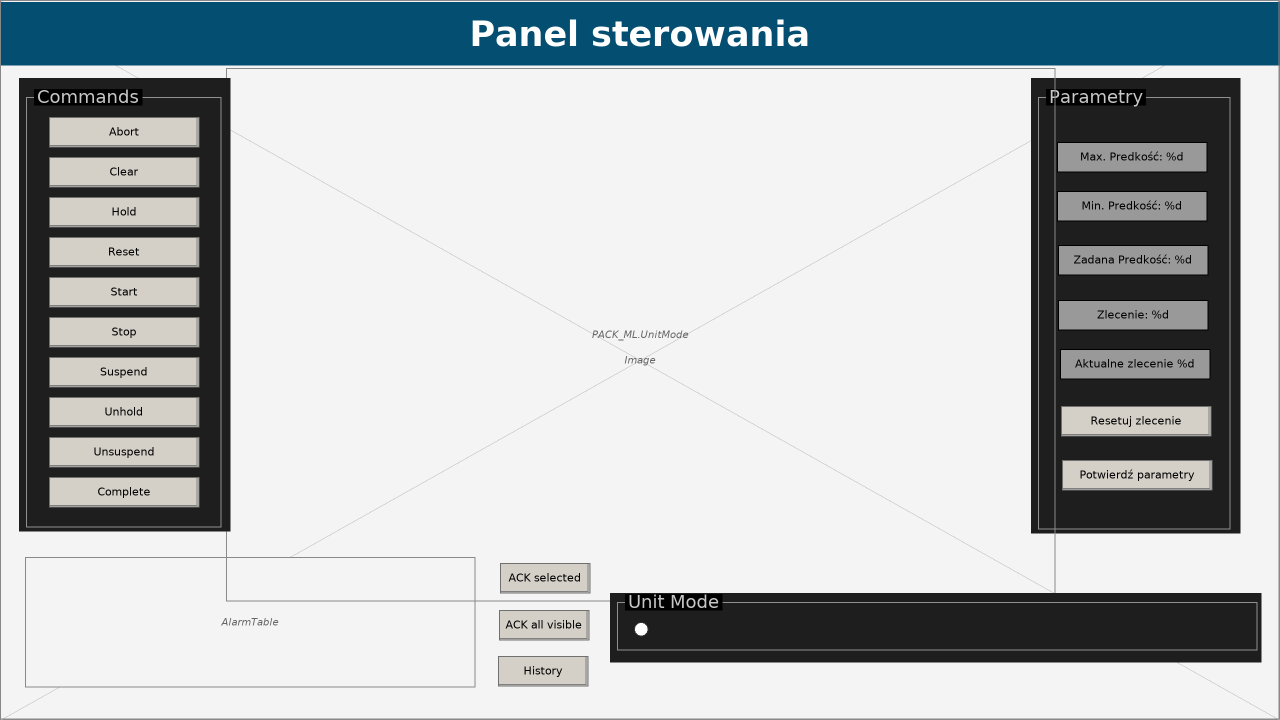
VISUALIZATION Panel  // 1280x720
VAR_IN_OUT
END_VAR
VAR
	bAckSel : BOOL;
	bAckVisible : BOOL;
	bHistory : BOOL;
	bFreezeScrlPos : BOOL;
END_VAR
    Image (0,0 1280x720)
    Rectangle (0,2 1280x63), "Panel sterowania"
    AlarmTable (25,557 450x130)
        p1521930926: __All
        p1663851261: __All
        p428520879: bAckSel
        p2607059081: bAckVisible
        p3266827225: bHistory
        p3894972949: bFreezeScrlPos
    Button (500,563 90x30), "ACK selected"
        toggle bAckSel
    Button (499,610 90x30), "ACK all visible"
        toggle bAckVisible
    Button (498,656 90x30), "History"
        toggle bHistory
    Rectangle (1031,78 209x455)
    GroupBox (1038,89 192x440), "Parametry"
        RoundedRectangle (19,53 150x30), "Max. Predkość: %d", text variable: PLC_PRG.iMaxPredkosc_visu, input disabled if: NOT ( PLC_PRG.unitModeManager.ActiveUnitMode.CurrentState = PACK_ML.Resetting )
            OnMouseClick: write PLC_PRG.iMaxPredkosc_visu via VisuDialogs.Numpad, min 0, max 10
        RoundedRectangle (19,102 150x30), "Min. Predkość: %d", text variable: PLC_PRG.iMInPredkosc_visu, input disabled if: NOT ( PLC_PRG.unitModeManager.ActiveUnitMode.CurrentState = PACK_ML.Resetting )
            OnMouseClick: write PLC_PRG.iMInPredkosc_visu via VisuDialogs.Numpad, min 0, max 10
        RoundedRectangle (20,156 150x30), "Zadana Predkość: %d", text variable: PLC_PRG.iPredkoscZadana_visu, input disabled if: NOT ( PLC_PRG.unitModeManager.ActiveUnitMode.CurrentState = PACK_ML.Resetting )
            OnMouseClick: write PLC_PRG.iPredkoscZadana_visu via VisuDialogs.Numpad, min 0, max 10
        RoundedRectangle (20,211 150x30), "Zlecenie: %d", text variable: PLC_PRG.iZlecenie_visu, input disabled if: NOT ( PLC_PRG.unitModeManager.ActiveUnitMode.CurrentState = PACK_ML.Resetting )
            OnMouseClick: write PLC_PRG.iZlecenie_visu via VisuDialogs.Numpad, min 0, max 100
        RoundedRectangle (22,260 150x30), "Aktualne zlecenie %d", text variable: PLC_PRG.iAktualnaLiczbaZleconychProduktow_visu
            OnMouseClick: write  via VisuDialogs.Numpad, min 0, max 10
        Button (23,317 150x30), "Resetuj zlecenie", input disabled if: NOT ( PLC_PRG.unitModeManager.ActiveUnitMode.CurrentState = PACK_ML.Resetting )
            tap PLC_PRG.xResetZlecenie_visu
            OnMouseClick:  
        Button (24,371 150x30), "Potwierdź parametry", input disabled if: NOT ( PLC_PRG.unitModeManager.ActiveUnitMode.CurrentState = PACK_ML.Resetting )
            tap PLC_PRG.xPotwierdzParametry_visu
            OnMouseClick:  
    Frame (226,68 829x533)
        shows PACK_ML.UnitMode(um := PLC_PRG.currentUnitMode)
    Rectangle (19,78 211x453)
    GroupBox (26,89 195x438), "Commands"
        Button (23,28 150x30), "Abort"
            tap PLC_PRG.xAbort
        Button (23,68 150x30), "Clear"
            tap PLC_PRG.xClear
        Button (23,108 150x30), "Hold"
            tap PLC_PRG.xHold
        Button (23,148 150x30), "Reset"
            tap PLC_PRG.xReset
        Button (23,188 150x30), "Start"
            tap PLC_PRG.xStart
        Button (23,228 150x30), "Stop"
            tap PLC_PRG.xStop
        Button (23,268 150x30), "Suspend"
            tap PLC_PRG.xSuspend
        Button (23,308 150x30), "Unhold"
            tap PLC_PRG.xUnHold
        Button (23,348 150x30), "Unsuspend"
            tap PLC_PRG.xUnSuspend
        Button (23,388 150x30), "Complete"
            tap PLC_PRG.xActingStateComplete
    Group (610,593 633x69)
        Rectangle (0,0 651x69)
        GroupBox (7,1 640x56), "Unit Mode"
        RadioButton (22,19 626x34), variable: PLC_PRG.iSelectedUnitMode
            Areas[0]: Text=Production
            Areas[1]: Text=Semi Auto Production
            Areas[2]: Text=Setup
END_VISUALIZATION

(* text list AlarmGroup1 (id | default)
  5 | Maszyna w stanie ABORTED
  4 | Maszyna w stanie SUSPENDED
  3 | Maszyna w stanie HELD
  2 | Koniec przerwy
  1 | Awaria czujnika wejściowego
  0 | Przycisk bezpieczeństwa
   |  *)

(* text list AlarmGroup2 (id | default)
   |  *)

(* text list AlarmGroup3 (id | default)
   |  *)

(* text list AlarmGroup (id | default)
   |  *)
